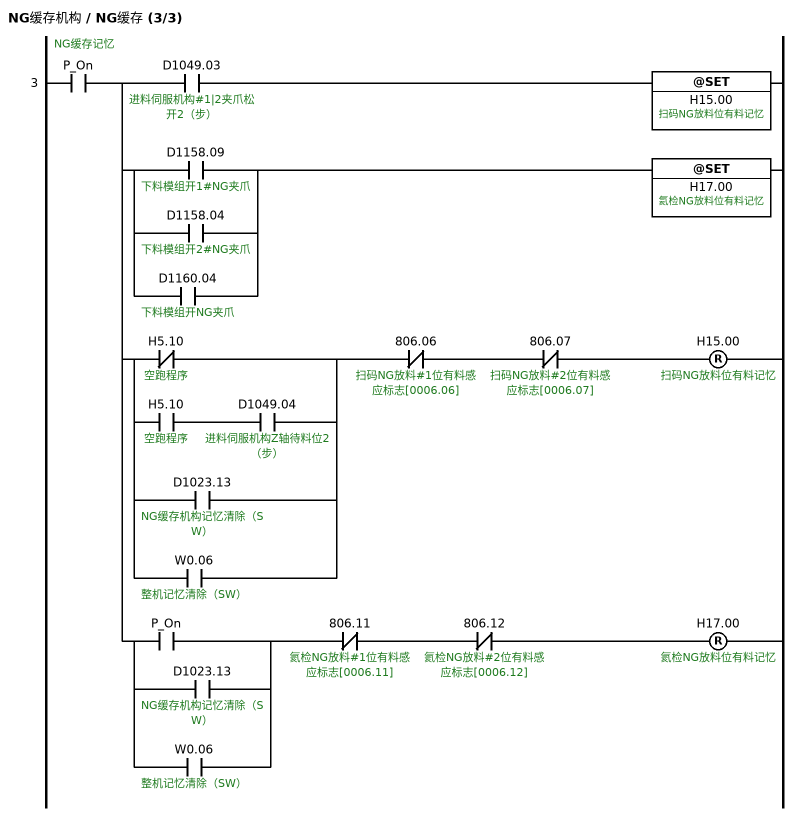
; rung 3: NG缓存记忆
LD P_On
OUT TR0
AND D1049.03  ; 进料伺服机构#1|2夹爪松开2（步）
@SET H15.00  ; 扫码NG放料位有料记忆
LD TR0
LD D1158.09  ; 下料模组开1#NG夹爪
OR D1158.04  ; 下料模组开2#NG夹爪
OR D1160.04  ; 下料模组开NG夹爪
ANDLD
@SET H17.00  ; 氦检NG放料位有料记忆
LD TR0
LDNOT H5.10  ; 空跑程序
LD H5.10  ; 空跑程序
AND D1049.04  ; 进料伺服机构Z轴待料位2（步）
ORLD
OR D1023.13  ; NG缓存机构记忆清除（SW）
OR W0.06  ; 整机记忆清除（SW）
ANDLD
ANDNOT 806.06  ; 扫码NG放料#1位有料感应标志[0006.06]
ANDNOT 806.07  ; 扫码NG放料#2位有料感应标志[0006.07]
RSET H15.00  ; 扫码NG放料位有料记忆
LD TR0
LD P_On
OR D1023.13  ; NG缓存机构记忆清除（SW）
OR W0.06  ; 整机记忆清除（SW）
ANDLD
ANDNOT 806.11  ; 氦检NG放料#1位有料感应标志[0006.11]
ANDNOT 806.12  ; 氦检NG放料#2位有料感应标志[0006.12]
RSET H17.00  ; 氦检NG放料位有料记忆

### Section 外部输出

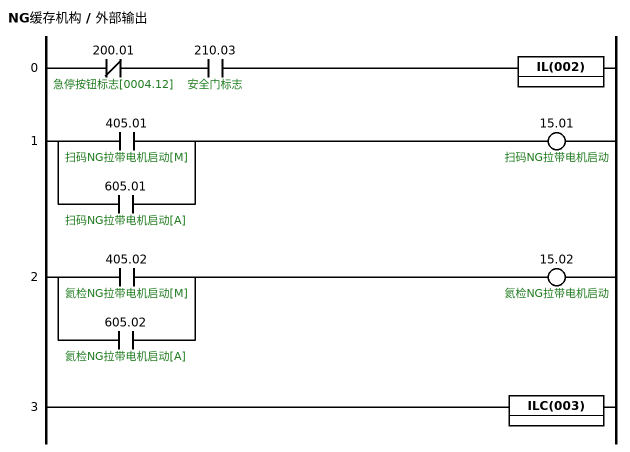
; rung 0
LDNOT 200.01  ; 急停按钮标志[0004.12]
AND 210.03  ; 安全门标志
IL(002)
; rung 1
LD 405.01  ; 扫码NG拉带电机启动[M]
OR 605.01  ; 扫码NG拉带电机启动[A]
OUT 15.01  ; 扫码NG拉带电机启动
; rung 2
LD 405.02  ; 氦检NG拉带电机启动[M]
OR 605.02  ; 氦检NG拉带电机启动[A]
OUT 15.02  ; 氦检NG拉带电机启动
; rung 3
ILC(003)

### Section END
; rung 0
END(001)

## Program Common (cyclic task 6)

### Section 动作延时

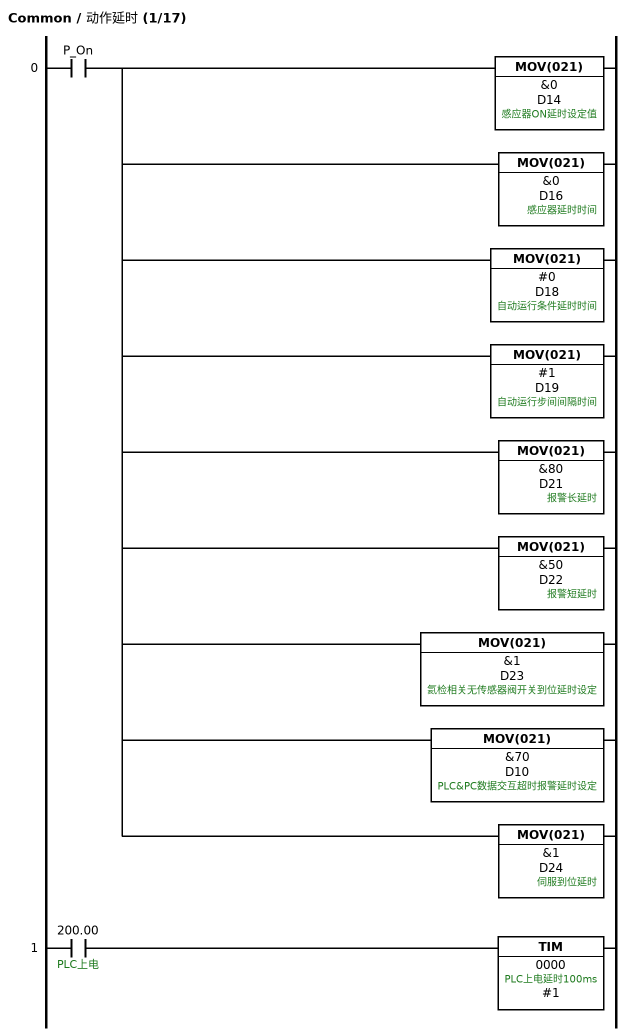
; rung 0
LD P_On
MOV(021) &0 D14  ; 感应器ON延时设定值
MOV(021) &0 D16  ; 感应器延时时间
MOV(021) #0 D18  ; 自动运行条件延时时间
MOV(021) #1 D19  ; 自动运行步间间隔时间
MOV(021) &80 D21  ; 报警长延时
MOV(021) &50 D22  ; 报警短延时
MOV(021) &1 D23  ; 氦检相关无传感器阀开关到位延时设定
MOV(021) &70 D10  ; PLC&PC数据交互超时报警延时设定
MOV(021) &1 D24  ; 伺服到位延时
; rung 1
LD 200.00  ; PLC上电
TIM 0000 #1  ; PLC上电延时100ms

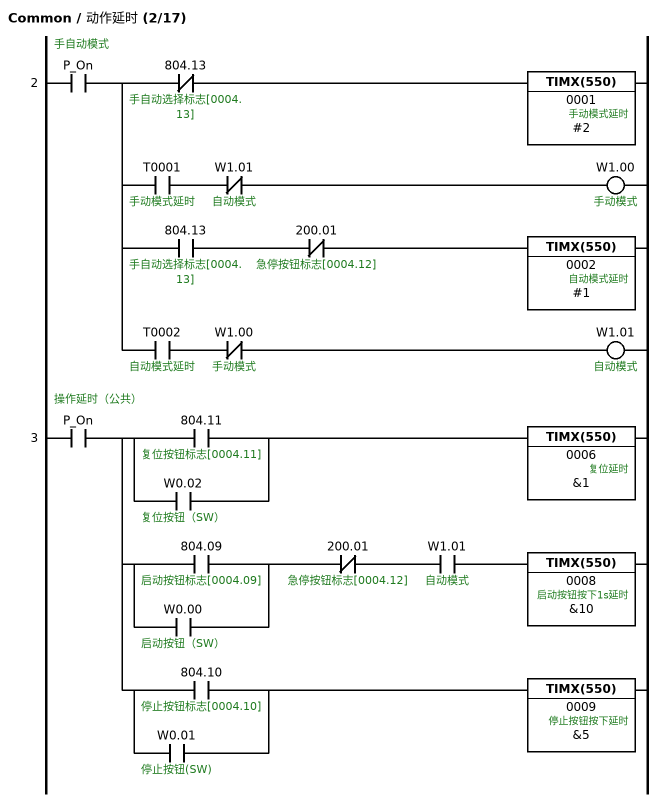
; rung 2: 手自动模式
LD P_On
OUT TR0
ANDNOT 804.13  ; 手自动选择标志[0004.13]
TIMX(550) 0001 #2  ; 手动模式延时
LD TR0
AND T0001  ; 手动模式延时
ANDNOT W1.01  ; 自动模式
OUT W1.00  ; 手动模式
LD TR0
AND 804.13  ; 手自动选择标志[0004.13]
ANDNOT 200.01  ; 急停按钮标志[0004.12]
TIMX(550) 0002 #1  ; 自动模式延时
LD TR0
AND T0002  ; 自动模式延时
ANDNOT W1.00  ; 手动模式
OUT W1.01  ; 自动模式
; rung 3: 操作延时（公共）
LD P_On
OUT TR0
LD 804.11  ; 复位按钮标志[0004.11]
OR W0.02  ; 复位按钮（SW）
ANDLD
TIMX(550) 0006 &1  ; 复位延时
LD TR0
LD 804.09  ; 启动按钮标志[0004.09]
OR W0.00  ; 启动按钮（SW）
ANDLD
ANDNOT 200.01  ; 急停按钮标志[0004.12]
AND W1.01  ; 自动模式
TIMX(550) 0008 &10  ; 启动按钮按下1s延时
LD TR0
LD 804.10  ; 停止按钮标志[0004.10]
OR W0.01  ; 停止按钮(SW)
ANDLD
TIMX(550) 0009 &5  ; 停止按钮按下延时

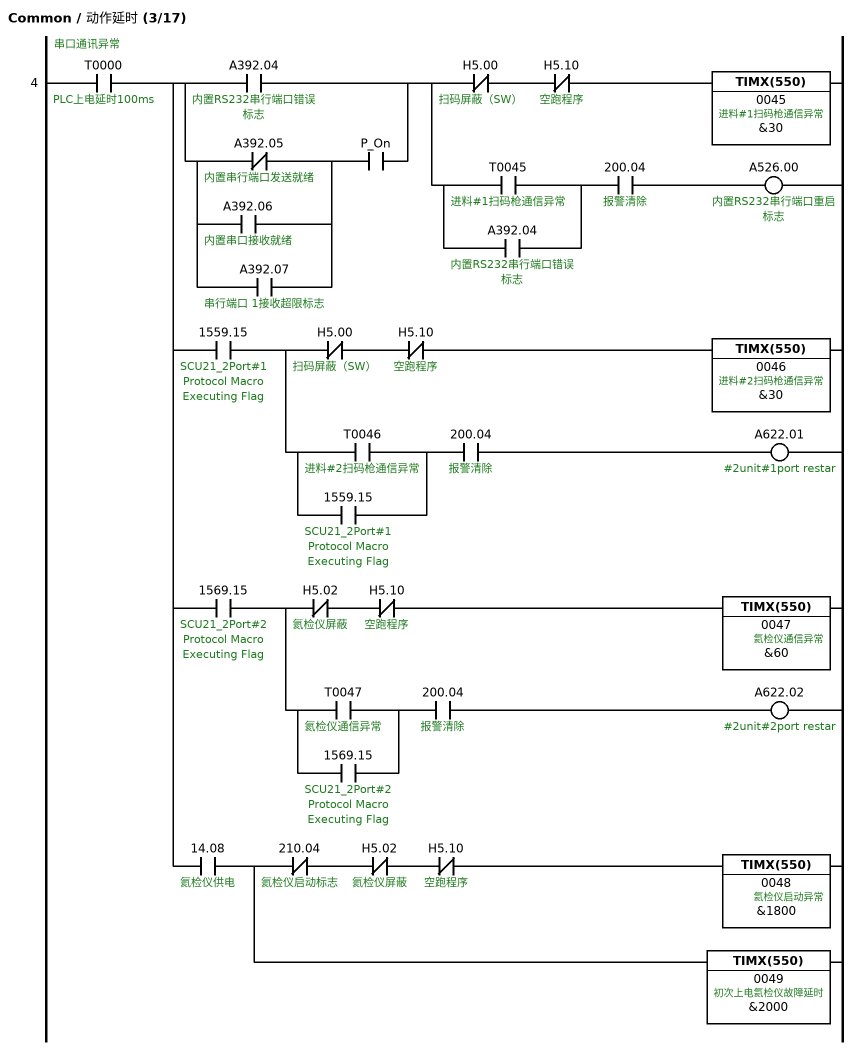
; rung 4: 串口通讯异常
LD T0000  ; PLC上电延时100ms
OUT TR0
LD A392.04  ; 内置RS232串行端口错误标志
LDNOT A392.05  ; 内置串行端口发送就绪
OR A392.06  ; 内置串口接收就绪
OR A392.07  ; 串行端口 1接收超限标志
AND P_On
ORLD
ANDLD
OUT TR1
ANDNOT H5.00  ; 扫码屏蔽（SW）
ANDNOT H5.10  ; 空跑程序
TIMX(550) 0045 &30  ; 进料#1扫码枪通信异常
LD TR1
LD T0045  ; 进料#1扫码枪通信异常
OR A392.04  ; 内置RS232串行端口错误标志
ANDLD
AND 200.04  ; 报警清除
OUT A526.00  ; 内置RS232串行端口重启标志
LD TR0
AND 1559.15  ; SCU21_2Port#1 Protocol Macro Executing Flag
OUT TR1
ANDNOT H5.00  ; 扫码屏蔽（SW）
ANDNOT H5.10  ; 空跑程序
TIMX(550) 0046 &30  ; 进料#2扫码枪通信异常
LD TR1
LD T0046  ; 进料#2扫码枪通信异常
OR 1559.15  ; SCU21_2Port#1 Protocol Macro Executing Flag
ANDLD
AND 200.04  ; 报警清除
OUT A622.01  ; #2unit#1port restar
LD TR0
AND 1569.15  ; SCU21_2Port#2 Protocol Macro Executing Flag
OUT TR1
ANDNOT H5.02  ; 氦检仪屏蔽
ANDNOT H5.10  ; 空跑程序
TIMX(550) 0047 &60  ; 氦检仪通信异常
LD TR1
LD T0047  ; 氦检仪通信异常
OR 1569.15  ; SCU21_2Port#2 Protocol Macro Executing Flag
ANDLD
AND 200.04  ; 报警清除
OUT A622.02  ; #2unit#2port restar
LD TR0
AND 14.08  ; 氦检仪供电
OUT TR0
ANDNOT 210.04  ; 氦检仪启动标志
ANDNOT H5.02  ; 氦检仪屏蔽
ANDNOT H5.10  ; 空跑程序
TIMX(550) 0048 &1800  ; 氦检仪启动异常
LD TR0
TIMX(550) 0049 &2000  ; 初次上电氦检仪故障延时
; rung 5: AI断线检测

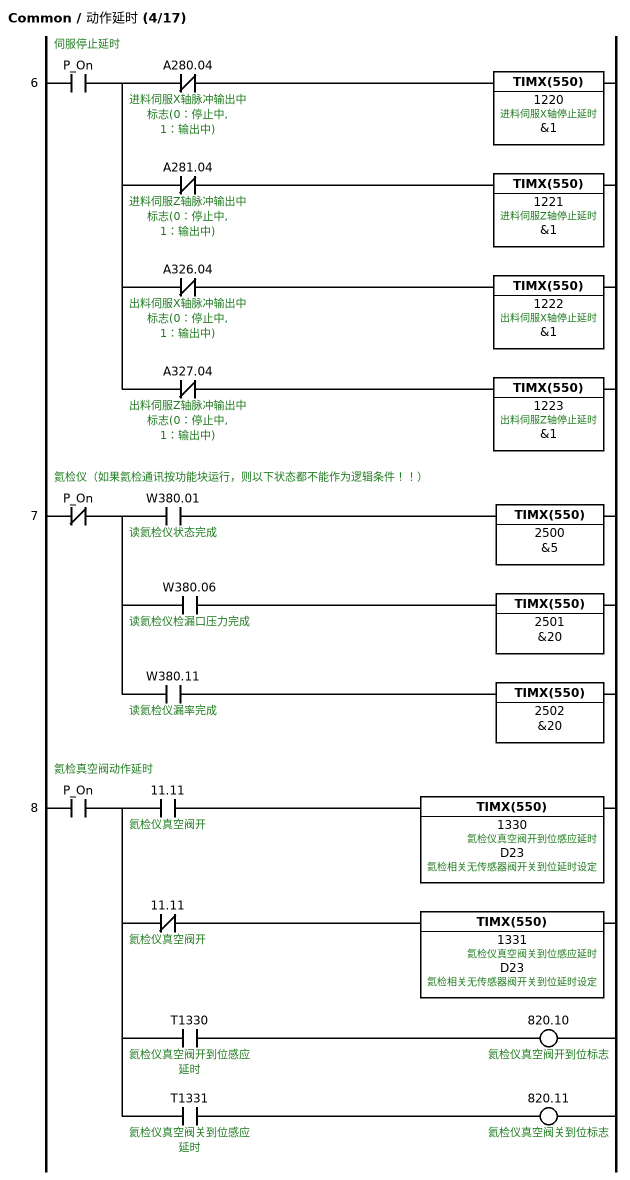
; rung 6: 伺服停止延时
LD P_On
OUT TR0
ANDNOT A280.04  ; 进料伺服X轴脉冲输出中标志(0：停止中,1：输出中)
TIMX(550) 1220 &1  ; 进料伺服X轴停止延时
LD TR0
ANDNOT A281.04  ; 进料伺服Z轴脉冲输出中标志(0：停止中,1：输出中)
TIMX(550) 1221 &1  ; 进料伺服Z轴停止延时
LD TR0
ANDNOT A326.04  ; 出料伺服X轴脉冲输出中标志(0：停止中,1：输出中)
TIMX(550) 1222 &1  ; 出料伺服X轴停止延时
LD TR0
ANDNOT A327.04  ; 出料伺服Z轴脉冲输出中标志(0：停止中,1：输出中)
TIMX(550) 1223 &1  ; 出料伺服Z轴停止延时
; rung 7: 氦检仪（如果氦检通讯按功能块运行，则以下状态都不能作为逻辑条件！！）
LDNOT P_On
OUT TR0
AND W380.01  ; 读氦检仪状态完成
TIMX(550) 2500 &5
LD TR0
AND W380.06  ; 读氦检仪检漏口压力完成
TIMX(550) 2501 &20
LD TR0
AND W380.11  ; 读氦检仪漏率完成
TIMX(550) 2502 &20
; rung 8: 氦检真空阀动作延时
LD P_On
OUT TR0
AND 11.11  ; 氦检仪真空阀开
TIMX(550) 1330 D23  ; 氦检相关无传感器阀开关到位延时设定, 氦检仪真空阀开到位感应延时
LD TR0
ANDNOT 11.11  ; 氦检仪真空阀开
TIMX(550) 1331 D23  ; 氦检相关无传感器阀开关到位延时设定, 氦检仪真空阀关到位感应延时
LD TR0
AND T1330  ; 氦检仪真空阀开到位感应延时
OUT 820.10  ; 氦检仪真空阀开到位标志
LD TR0
AND T1331  ; 氦检仪真空阀关到位感应延时
OUT 820.11  ; 氦检仪真空阀关到位标志

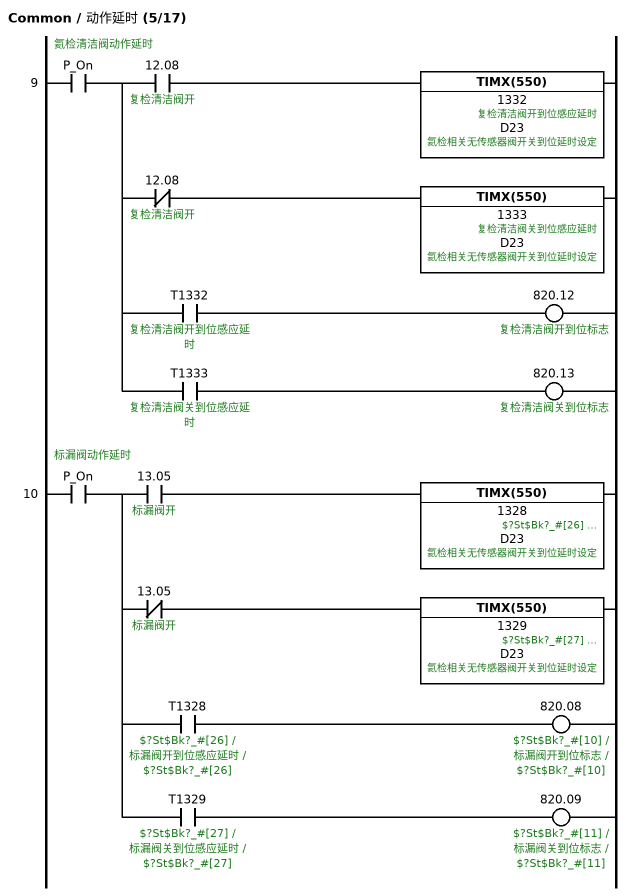
; rung 9: 氦检清洁阀动作延时
LD P_On
OUT TR0
AND 12.08  ; 复检清洁阀开
TIMX(550) 1332 D23  ; 氦检相关无传感器阀开关到位延时设定, 复检清洁阀开到位感应延时
LD TR0
ANDNOT 12.08  ; 复检清洁阀开
TIMX(550) 1333 D23  ; 氦检相关无传感器阀开关到位延时设定, 复检清洁阀关到位感应延时
LD TR0
AND T1332  ; 复检清洁阀开到位感应延时
OUT 820.12  ; 复检清洁阀开到位标志
LD TR0
AND T1333  ; 复检清洁阀关到位感应延时
OUT 820.13  ; 复检清洁阀关到位标志
; rung 10: 标漏阀动作延时
LD P_On
OUT TR0
AND 13.05  ; 标漏阀开
TIMX(550) 1328 D23  ; 氦检相关无传感器阀开关到位延时设定, $?St$Bk?_#[26] / 标漏阀开到位感应延时 / $?St$Bk?_#[26]
LD TR0
ANDNOT 13.05  ; 标漏阀开
TIMX(550) 1329 D23  ; 氦检相关无传感器阀开关到位延时设定, $?St$Bk?_#[27] / 标漏阀关到位感应延时 / $?St$Bk?_#[27]
LD TR0
AND T1328  ; $?St$Bk?_#[26] / 标漏阀开到位感应延时 / $?St$Bk?_#[26]
OUT 820.08  ; $?St$Bk?_#[10] / 标漏阀开到位标志 / $?St$Bk?_#[10]
LD TR0
AND T1329  ; $?St$Bk?_#[27] / 标漏阀关到位感应延时 / $?St$Bk?_#[27]
OUT 820.09  ; $?St$Bk?_#[11] / 标漏阀关到位标志 / $?St$Bk?_#[11]

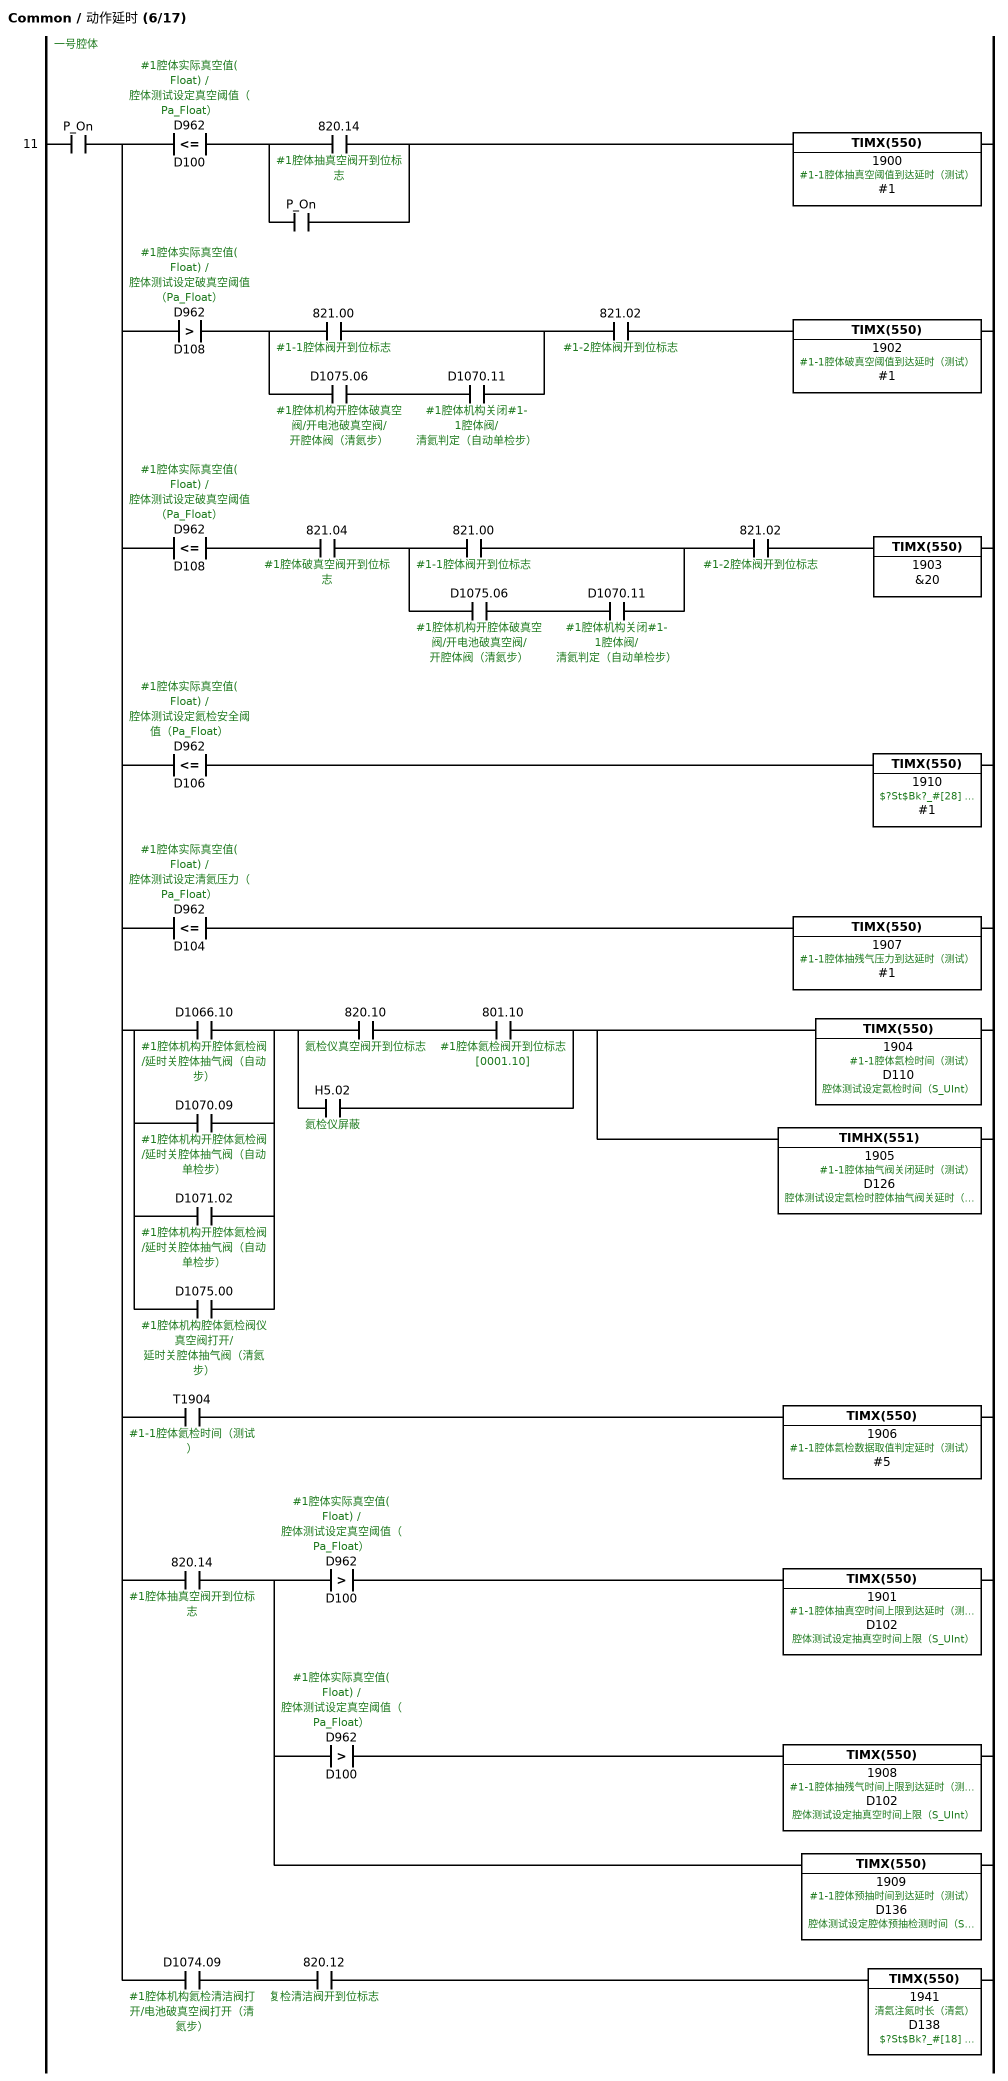
; rung 11: 一号腔体
LD P_On
OUT TR0
AND<=F(332) D962 D100  ; #1腔体实际真空值(Float), 腔体测试设定真空阈值（Pa_Float）
LD 820.14  ; #1腔体抽真空阀开到位标志
OR P_On
ANDLD
TIMX(550) 1900 #1  ; #1-1腔体抽真空阈值到达延时（测试）
LD TR0
AND>F(333) D962 D108  ; #1腔体实际真空值(Float), 腔体测试设定破真空阈值（Pa_Float）
LD 821.00  ; #1-1腔体阀开到位标志
LD D1075.06  ; #1腔体机构开腔体破真空阀/开电池破真空阀/开腔体阀（清氦步）
AND D1070.11  ; #1腔体机构关闭#1-1腔体阀/清氦判定（自动单检步）
ORLD
ANDLD
AND 821.02  ; #1-2腔体阀开到位标志
TIMX(550) 1902 #1  ; #1-1腔体破真空阈值到达延时（测试）
LD TR0
AND<=F(332) D962 D108  ; #1腔体实际真空值(Float), 腔体测试设定破真空阈值（Pa_Float）
AND 821.04  ; #1腔体破真空阀开到位标志
LD 821.00  ; #1-1腔体阀开到位标志
LD D1075.06  ; #1腔体机构开腔体破真空阀/开电池破真空阀/开腔体阀（清氦步）
AND D1070.11  ; #1腔体机构关闭#1-1腔体阀/清氦判定（自动单检步）
ORLD
ANDLD
AND 821.02  ; #1-2腔体阀开到位标志
TIMX(550) 1903 &20
LD TR0
AND<=F(332) D962 D106  ; #1腔体实际真空值(Float), 腔体测试设定氦检安全阈值（Pa_Float）
TIMX(550) 1910 #1  ; $?St$Bk?_#[28] / #1-1腔体真空在可氦检状态（测试） / $?St$Bk?_#[28]
LD TR0
AND<=F(332) D962 D104  ; #1腔体实际真空值(Float), 腔体测试设定清氦压力（Pa_Float）
TIMX(550) 1907 #1  ; #1-1腔体抽残气压力到达延时（测试）
LD TR0
LD D1066.10  ; #1腔体机构开腔体氦检阀/延时关腔体抽气阀（自动步）
OR D1070.09  ; #1腔体机构开腔体氦检阀/延时关腔体抽气阀（自动单检步）
OR D1071.02  ; #1腔体机构开腔体氦检阀/延时关腔体抽气阀（自动单检步）
OR D1075.00  ; #1腔体机构腔体氦检阀仪真空阀打开/延时关腔体抽气阀（清氦步）
ANDLD
LD 820.10  ; 氦检仪真空阀开到位标志
AND 801.10  ; #1腔体氦检阀开到位标志[0001.10]
OR H5.02  ; 氦检仪屏蔽
ANDLD
TIMX(550) 1904 D110  ; 腔体测试设定氦检时间（S_UInt）, #1-1腔体氦检时间（测试）
TIMHX(551) 1905 D126  ; 腔体测试设定氦检时腔体抽气阀关延时（S_UInt）, #1-1腔体抽气阀关闭延时（测试）
LD TR0
AND T1904  ; #1-1腔体氦检时间（测试）
TIMX(550) 1906 #5  ; #1-1腔体氦检数据取值判定延时（测试）
LD TR0
AND 820.14  ; #1腔体抽真空阀开到位标志
OUT TR1
AND>F(333) D962 D100  ; #1腔体实际真空值(Float), 腔体测试设定真空阈值（Pa_Float）
TIMX(550) 1901 D102  ; 腔体测试设定抽真空时间上限（S_UInt）, #1-1腔体抽真空时间上限到达延时（测试）
LD TR1
AND>F(333) D962 D100  ; #1腔体实际真空值(Float), 腔体测试设定真空阈值（Pa_Float）
TIMX(550) 1908 D102  ; 腔体测试设定抽真空时间上限（S_UInt）, #1-1腔体抽残气时间上限到达延时（测试）
LD TR1
TIMX(550) 1909 D136  ; 腔体测试设定腔体预抽检测时间（S_UInt）, #1-1腔体预抽时间到达延时（测试）
LD TR0
AND D1074.09  ; #1腔体机构氦检清洁阀打开/电池破真空阀打开（清氦步）
AND 820.12  ; 复检清洁阀开到位标志
TIMX(550) 1941 D138  ; $?St$Bk?_#[18] / 管路清氦注氮时间（S_UInt） / $?St$Bk?_#[18], 清氦注氮时长（清氦）

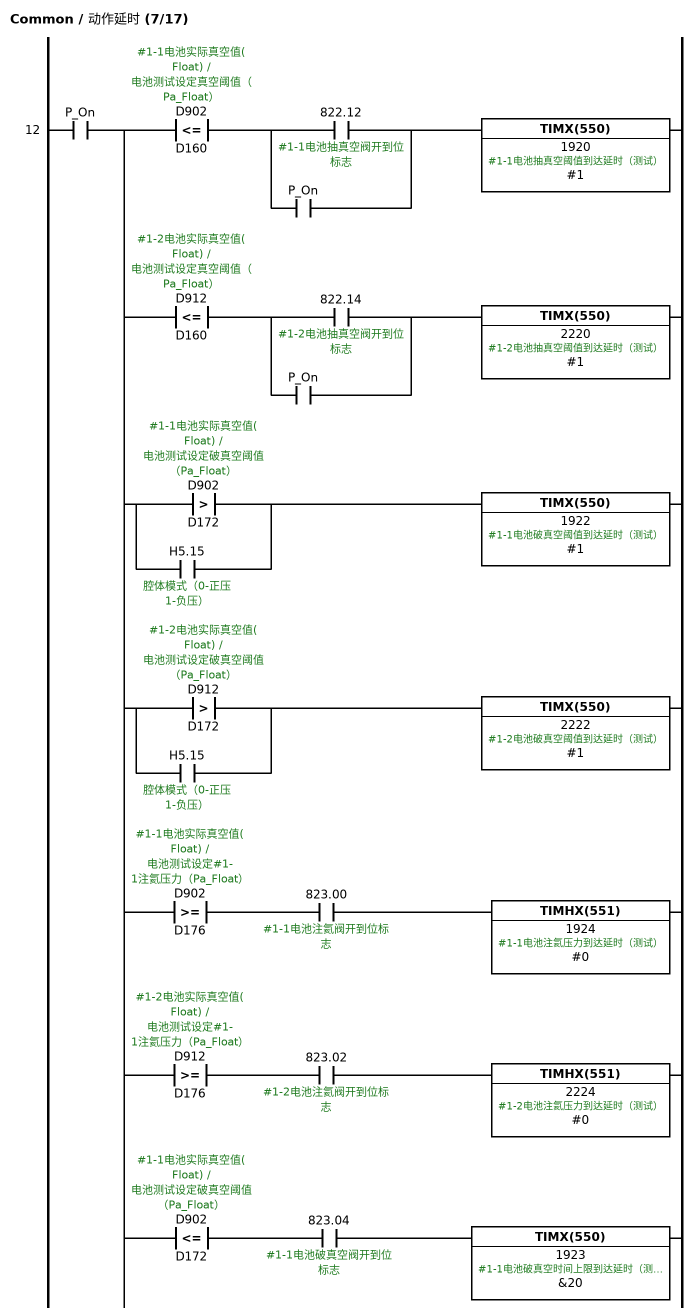

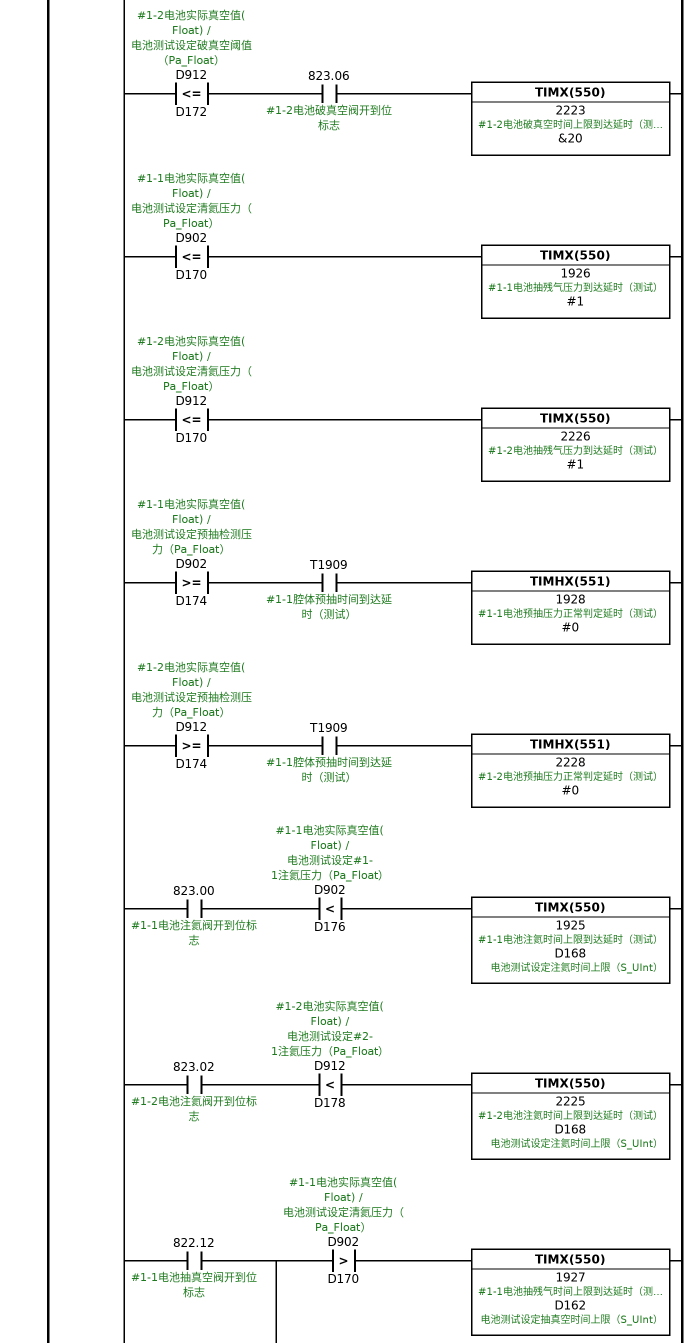

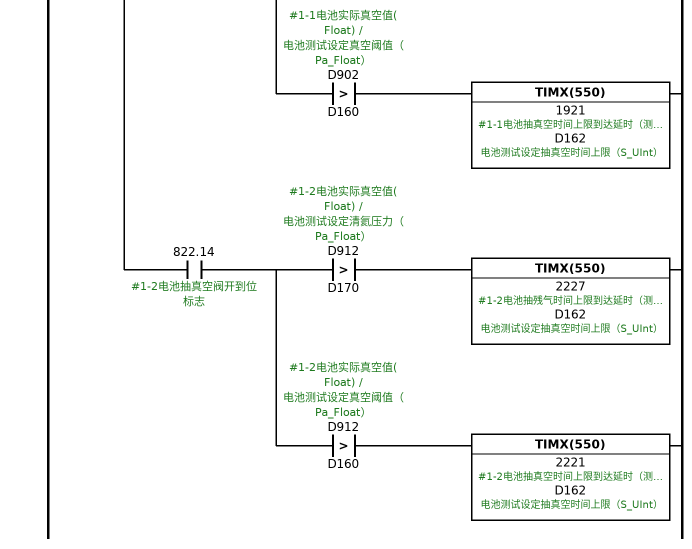
; rung 12
LD P_On
OUT TR0
AND<=F(332) D902 D160  ; #1-1电池实际真空值(Float), 电池测试设定真空阈值（Pa_Float）
LD 822.12  ; #1-1电池抽真空阀开到位标志
OR P_On
ANDLD
TIMX(550) 1920 #1  ; #1-1电池抽真空阈值到达延时（测试）
LD TR0
AND<=F(332) D912 D160  ; #1-2电池实际真空值(Float), 电池测试设定真空阈值（Pa_Float）
LD 822.14  ; #1-2电池抽真空阀开到位标志
OR P_On
ANDLD
TIMX(550) 2220 #1  ; #1-2电池抽真空阈值到达延时（测试）
LD TR0
LD>F(333) D902 D172  ; #1-1电池实际真空值(Float), 电池测试设定破真空阈值（Pa_Float）
OR H5.15  ; 腔体模式（0-正压 1-负压）
ANDLD
TIMX(550) 1922 #1  ; #1-1电池破真空阈值到达延时（测试）
LD TR0
LD>F(333) D912 D172  ; #1-2电池实际真空值(Float), 电池测试设定破真空阈值（Pa_Float）
OR H5.15  ; 腔体模式（0-正压 1-负压）
ANDLD
TIMX(550) 2222 #1  ; #1-2电池破真空阈值到达延时（测试）
LD TR0
AND>=F(334) D902 D176  ; #1-1电池实际真空值(Float), 电池测试设定#1-1注氦压力（Pa_Float）
AND 823.00  ; #1-1电池注氦阀开到位标志
TIMHX(551) 1924 #0  ; #1-1电池注氦压力到达延时（测试）
LD TR0
AND>=F(334) D912 D176  ; #1-2电池实际真空值(Float), 电池测试设定#1-1注氦压力（Pa_Float）
AND 823.02  ; #1-2电池注氦阀开到位标志
TIMHX(551) 2224 #0  ; #1-2电池注氦压力到达延时（测试）
LD TR0
AND<=F(332) D902 D172  ; #1-1电池实际真空值(Float), 电池测试设定破真空阈值（Pa_Float）
AND 823.04  ; #1-1电池破真空阀开到位标志
TIMX(550) 1923 &20  ; #1-1电池破真空时间上限到达延时（测试）
LD TR0
AND<=F(332) D912 D172  ; #1-2电池实际真空值(Float), 电池测试设定破真空阈值（Pa_Float）
AND 823.06  ; #1-2电池破真空阀开到位标志
TIMX(550) 2223 &20  ; #1-2电池破真空时间上限到达延时（测试）
LD TR0
AND<=F(332) D902 D170  ; #1-1电池实际真空值(Float), 电池测试设定清氦压力（Pa_Float）
TIMX(550) 1926 #1  ; #1-1电池抽残气压力到达延时（测试）
LD TR0
AND<=F(332) D912 D170  ; #1-2电池实际真空值(Float), 电池测试设定清氦压力（Pa_Float）
TIMX(550) 2226 #1  ; #1-2电池抽残气压力到达延时（测试）
LD TR0
AND>=F(334) D902 D174  ; #1-1电池实际真空值(Float), 电池测试设定预抽检测压力（Pa_Float）
AND T1909  ; #1-1腔体预抽时间到达延时（测试）
TIMHX(551) 1928 #0  ; #1-1电池预抽压力正常判定延时（测试）
LD TR0
AND>=F(334) D912 D174  ; #1-2电池实际真空值(Float), 电池测试设定预抽检测压力（Pa_Float）
AND T1909  ; #1-1腔体预抽时间到达延时（测试）
TIMHX(551) 2228 #0  ; #1-2电池预抽压力正常判定延时（测试）
LD TR0
AND 823.00  ; #1-1电池注氦阀开到位标志
AND<F(331) D902 D176  ; #1-1电池实际真空值(Float), 电池测试设定#1-1注氦压力（Pa_Float）
TIMX(550) 1925 D168  ; 电池测试设定注氦时间上限（S_UInt）, #1-1电池注氦时间上限到达延时（测试）
LD TR0
AND 823.02  ; #1-2电池注氦阀开到位标志
AND<F(331) D912 D178  ; #1-2电池实际真空值(Float), 电池测试设定#2-1注氦压力（Pa_Float）
TIMX(550) 2225 D168  ; 电池测试设定注氦时间上限（S_UInt）, #1-2电池注氦时间上限到达延时（测试）
LD TR0
AND 822.12  ; #1-1电池抽真空阀开到位标志
OUT TR1
AND>F(333) D902 D170  ; #1-1电池实际真空值(Float), 电池测试设定清氦压力（Pa_Float）
TIMX(550) 1927 D162  ; 电池测试设定抽真空时间上限（S_UInt）, #1-1电池抽残气时间上限到达延时（测试）
LD TR1
AND>F(333) D902 D160  ; #1-1电池实际真空值(Float), 电池测试设定真空阈值（Pa_Float）
TIMX(550) 1921 D162  ; 电池测试设定抽真空时间上限（S_UInt）, #1-1电池抽真空时间上限到达延时（测试）
LD TR0
AND 822.14  ; #1-2电池抽真空阀开到位标志
OUT TR0
AND>F(333) D912 D170  ; #1-2电池实际真空值(Float), 电池测试设定清氦压力（Pa_Float）
TIMX(550) 2227 D162  ; 电池测试设定抽真空时间上限（S_UInt）, #1-2电池抽残气时间上限到达延时（测试）
LD TR0
AND>F(333) D912 D160  ; #1-2电池实际真空值(Float), 电池测试设定真空阈值（Pa_Float）
TIMX(550) 2221 D162  ; 电池测试设定抽真空时间上限（S_UInt）, #1-2电池抽真空时间上限到达延时（测试）

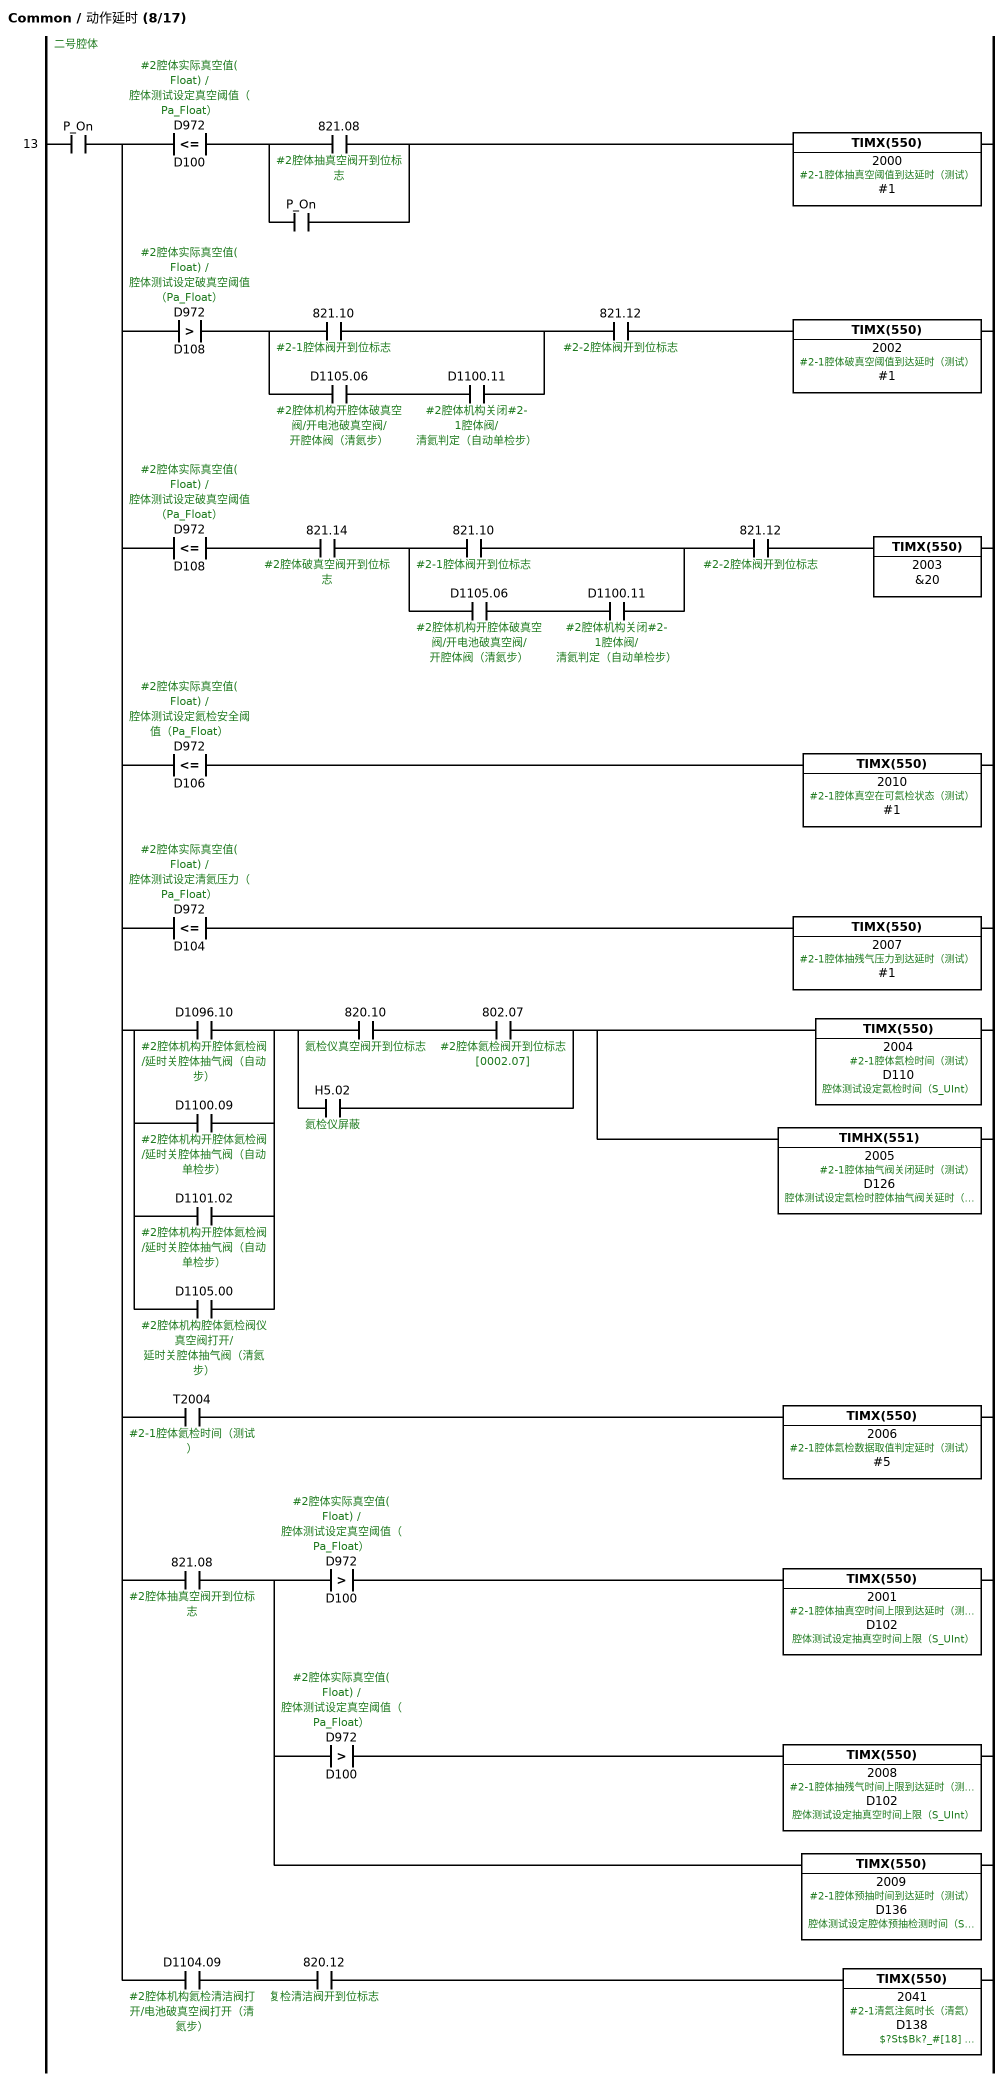
; rung 13: 二号腔体
LD P_On
OUT TR0
AND<=F(332) D972 D100  ; #2腔体实际真空值(Float), 腔体测试设定真空阈值（Pa_Float）
LD 821.08  ; #2腔体抽真空阀开到位标志
OR P_On
ANDLD
TIMX(550) 2000 #1  ; #2-1腔体抽真空阈值到达延时（测试）
LD TR0
AND>F(333) D972 D108  ; #2腔体实际真空值(Float), 腔体测试设定破真空阈值（Pa_Float）
LD 821.10  ; #2-1腔体阀开到位标志
LD D1105.06  ; #2腔体机构开腔体破真空阀/开电池破真空阀/开腔体阀（清氦步）
AND D1100.11  ; #2腔体机构关闭#2-1腔体阀/清氦判定（自动单检步）
ORLD
ANDLD
AND 821.12  ; #2-2腔体阀开到位标志
TIMX(550) 2002 #1  ; #2-1腔体破真空阈值到达延时（测试）
LD TR0
AND<=F(332) D972 D108  ; #2腔体实际真空值(Float), 腔体测试设定破真空阈值（Pa_Float）
AND 821.14  ; #2腔体破真空阀开到位标志
LD 821.10  ; #2-1腔体阀开到位标志
LD D1105.06  ; #2腔体机构开腔体破真空阀/开电池破真空阀/开腔体阀（清氦步）
AND D1100.11  ; #2腔体机构关闭#2-1腔体阀/清氦判定（自动单检步）
ORLD
ANDLD
AND 821.12  ; #2-2腔体阀开到位标志
TIMX(550) 2003 &20
LD TR0
AND<=F(332) D972 D106  ; #2腔体实际真空值(Float), 腔体测试设定氦检安全阈值（Pa_Float）
TIMX(550) 2010 #1  ; #2-1腔体真空在可氦检状态（测试）
LD TR0
AND<=F(332) D972 D104  ; #2腔体实际真空值(Float), 腔体测试设定清氦压力（Pa_Float）
TIMX(550) 2007 #1  ; #2-1腔体抽残气压力到达延时（测试）
LD TR0
LD D1096.10  ; #2腔体机构开腔体氦检阀/延时关腔体抽气阀（自动步）
OR D1100.09  ; #2腔体机构开腔体氦检阀/延时关腔体抽气阀（自动单检步）
OR D1101.02  ; #2腔体机构开腔体氦检阀/延时关腔体抽气阀（自动单检步）
OR D1105.00  ; #2腔体机构腔体氦检阀仪真空阀打开/延时关腔体抽气阀（清氦步）
ANDLD
LD 820.10  ; 氦检仪真空阀开到位标志
AND 802.07  ; #2腔体氦检阀开到位标志[0002.07]
OR H5.02  ; 氦检仪屏蔽
ANDLD
TIMX(550) 2004 D110  ; 腔体测试设定氦检时间（S_UInt）, #2-1腔体氦检时间（测试）
TIMHX(551) 2005 D126  ; 腔体测试设定氦检时腔体抽气阀关延时（S_UInt）, #2-1腔体抽气阀关闭延时（测试）
LD TR0
AND T2004  ; #2-1腔体氦检时间（测试）
TIMX(550) 2006 #5  ; #2-1腔体氦检数据取值判定延时（测试）
LD TR0
AND 821.08  ; #2腔体抽真空阀开到位标志
OUT TR1
AND>F(333) D972 D100  ; #2腔体实际真空值(Float), 腔体测试设定真空阈值（Pa_Float）
TIMX(550) 2001 D102  ; 腔体测试设定抽真空时间上限（S_UInt）, #2-1腔体抽真空时间上限到达延时（测试）
LD TR1
AND>F(333) D972 D100  ; #2腔体实际真空值(Float), 腔体测试设定真空阈值（Pa_Float）
TIMX(550) 2008 D102  ; 腔体测试设定抽真空时间上限（S_UInt）, #2-1腔体抽残气时间上限到达延时（测试）
LD TR1
TIMX(550) 2009 D136  ; 腔体测试设定腔体预抽检测时间（S_UInt）, #2-1腔体预抽时间到达延时（测试）
LD TR0
AND D1104.09  ; #2腔体机构氦检清洁阀打开/电池破真空阀打开（清氦步）
AND 820.12  ; 复检清洁阀开到位标志
TIMX(550) 2041 D138  ; $?St$Bk?_#[18] / 管路清氦注氮时间（S_UInt） / $?St$Bk?_#[18], #2-1清氦注氮时长（清氦）

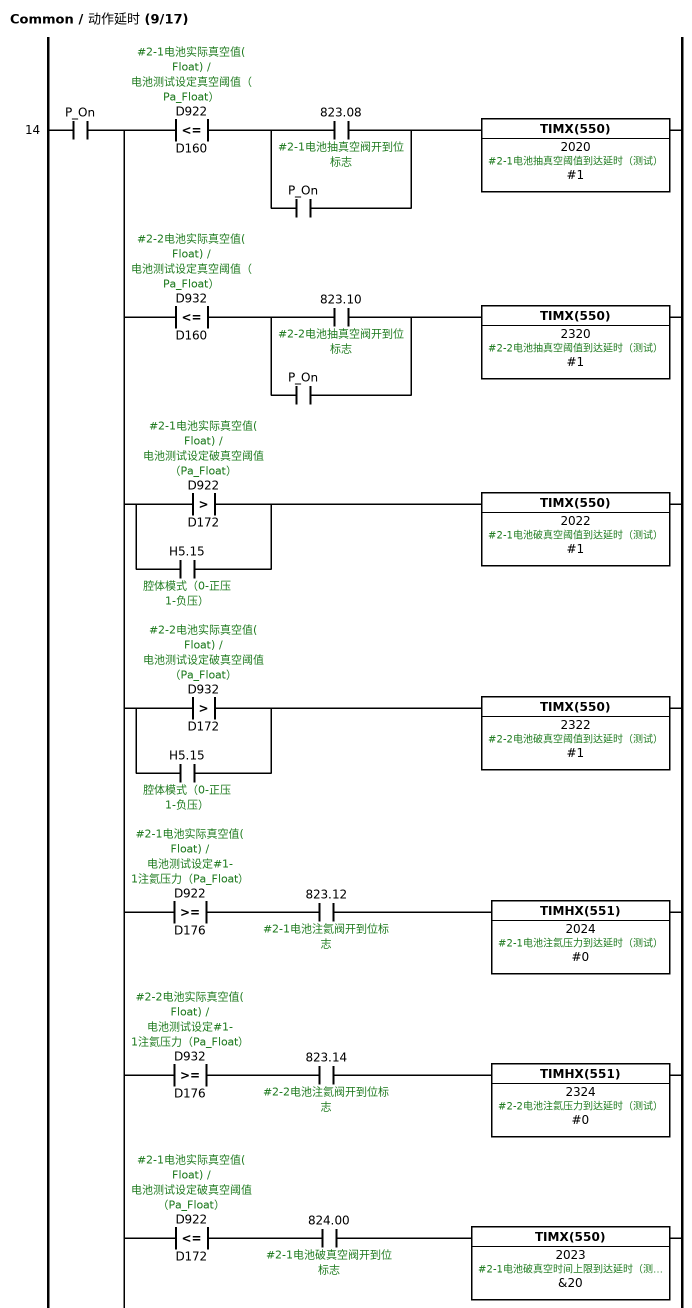

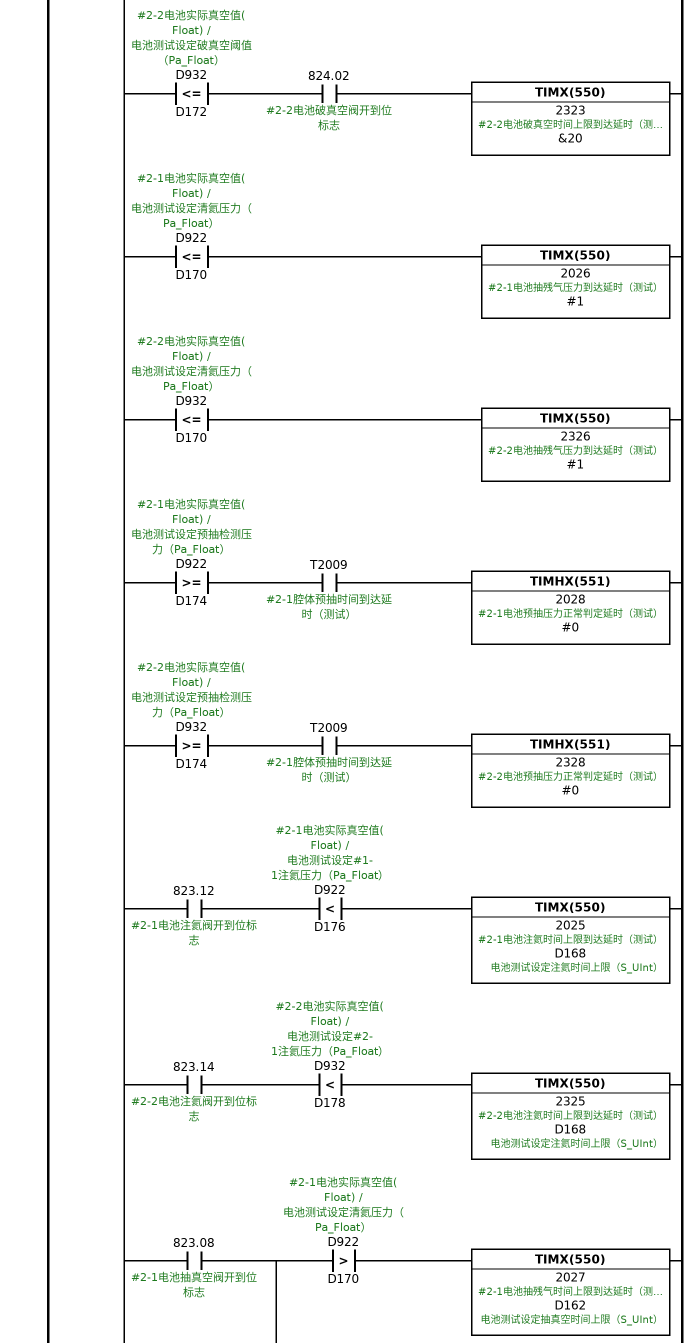

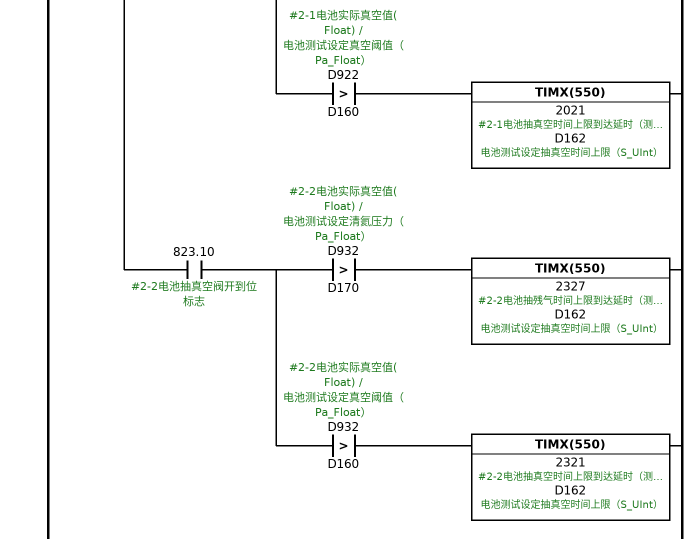
; rung 14
LD P_On
OUT TR0
AND<=F(332) D922 D160  ; #2-1电池实际真空值(Float), 电池测试设定真空阈值（Pa_Float）
LD 823.08  ; #2-1电池抽真空阀开到位标志
OR P_On
ANDLD
TIMX(550) 2020 #1  ; #2-1电池抽真空阈值到达延时（测试）
LD TR0
AND<=F(332) D932 D160  ; #2-2电池实际真空值(Float), 电池测试设定真空阈值（Pa_Float）
LD 823.10  ; #2-2电池抽真空阀开到位标志
OR P_On
ANDLD
TIMX(550) 2320 #1  ; #2-2电池抽真空阈值到达延时（测试）
LD TR0
LD>F(333) D922 D172  ; #2-1电池实际真空值(Float), 电池测试设定破真空阈值（Pa_Float）
OR H5.15  ; 腔体模式（0-正压 1-负压）
ANDLD
TIMX(550) 2022 #1  ; #2-1电池破真空阈值到达延时（测试）
LD TR0
LD>F(333) D932 D172  ; #2-2电池实际真空值(Float), 电池测试设定破真空阈值（Pa_Float）
OR H5.15  ; 腔体模式（0-正压 1-负压）
ANDLD
TIMX(550) 2322 #1  ; #2-2电池破真空阈值到达延时（测试）
LD TR0
AND>=F(334) D922 D176  ; #2-1电池实际真空值(Float), 电池测试设定#1-1注氦压力（Pa_Float）
AND 823.12  ; #2-1电池注氦阀开到位标志
TIMHX(551) 2024 #0  ; #2-1电池注氦压力到达延时（测试）
LD TR0
AND>=F(334) D932 D176  ; #2-2电池实际真空值(Float), 电池测试设定#1-1注氦压力（Pa_Float）
AND 823.14  ; #2-2电池注氦阀开到位标志
TIMHX(551) 2324 #0  ; #2-2电池注氦压力到达延时（测试）
LD TR0
AND<=F(332) D922 D172  ; #2-1电池实际真空值(Float), 电池测试设定破真空阈值（Pa_Float）
AND 824.00  ; #2-1电池破真空阀开到位标志
TIMX(550) 2023 &20  ; #2-1电池破真空时间上限到达延时（测试）
LD TR0
AND<=F(332) D932 D172  ; #2-2电池实际真空值(Float), 电池测试设定破真空阈值（Pa_Float）
AND 824.02  ; #2-2电池破真空阀开到位标志
TIMX(550) 2323 &20  ; #2-2电池破真空时间上限到达延时（测试）
LD TR0
AND<=F(332) D922 D170  ; #2-1电池实际真空值(Float), 电池测试设定清氦压力（Pa_Float）
TIMX(550) 2026 #1  ; #2-1电池抽残气压力到达延时（测试）
LD TR0
AND<=F(332) D932 D170  ; #2-2电池实际真空值(Float), 电池测试设定清氦压力（Pa_Float）
TIMX(550) 2326 #1  ; #2-2电池抽残气压力到达延时（测试）
LD TR0
AND>=F(334) D922 D174  ; #2-1电池实际真空值(Float), 电池测试设定预抽检测压力（Pa_Float）
AND T2009  ; #2-1腔体预抽时间到达延时（测试）
TIMHX(551) 2028 #0  ; #2-1电池预抽压力正常判定延时（测试）
LD TR0
AND>=F(334) D932 D174  ; #2-2电池实际真空值(Float), 电池测试设定预抽检测压力（Pa_Float）
AND T2009  ; #2-1腔体预抽时间到达延时（测试）
TIMHX(551) 2328 #0  ; #2-2电池预抽压力正常判定延时（测试）
LD TR0
AND 823.12  ; #2-1电池注氦阀开到位标志
AND<F(331) D922 D176  ; #2-1电池实际真空值(Float), 电池测试设定#1-1注氦压力（Pa_Float）
TIMX(550) 2025 D168  ; 电池测试设定注氦时间上限（S_UInt）, #2-1电池注氦时间上限到达延时（测试）
LD TR0
AND 823.14  ; #2-2电池注氦阀开到位标志
AND<F(331) D932 D178  ; #2-2电池实际真空值(Float), 电池测试设定#2-1注氦压力（Pa_Float）
TIMX(550) 2325 D168  ; 电池测试设定注氦时间上限（S_UInt）, #2-2电池注氦时间上限到达延时（测试）
LD TR0
AND 823.08  ; #2-1电池抽真空阀开到位标志
OUT TR1
AND>F(333) D922 D170  ; #2-1电池实际真空值(Float), 电池测试设定清氦压力（Pa_Float）
TIMX(550) 2027 D162  ; 电池测试设定抽真空时间上限（S_UInt）, #2-1电池抽残气时间上限到达延时（测试）
LD TR1
AND>F(333) D922 D160  ; #2-1电池实际真空值(Float), 电池测试设定真空阈值（Pa_Float）
TIMX(550) 2021 D162  ; 电池测试设定抽真空时间上限（S_UInt）, #2-1电池抽真空时间上限到达延时（测试）
LD TR0
AND 823.10  ; #2-2电池抽真空阀开到位标志
OUT TR0
AND>F(333) D932 D170  ; #2-2电池实际真空值(Float), 电池测试设定清氦压力（Pa_Float）
TIMX(550) 2327 D162  ; 电池测试设定抽真空时间上限（S_UInt）, #2-2电池抽残气时间上限到达延时（测试）
LD TR0
AND>F(333) D932 D160  ; #2-2电池实际真空值(Float), 电池测试设定真空阈值（Pa_Float）
TIMX(550) 2321 D162  ; 电池测试设定抽真空时间上限（S_UInt）, #2-2电池抽真空时间上限到达延时（测试）

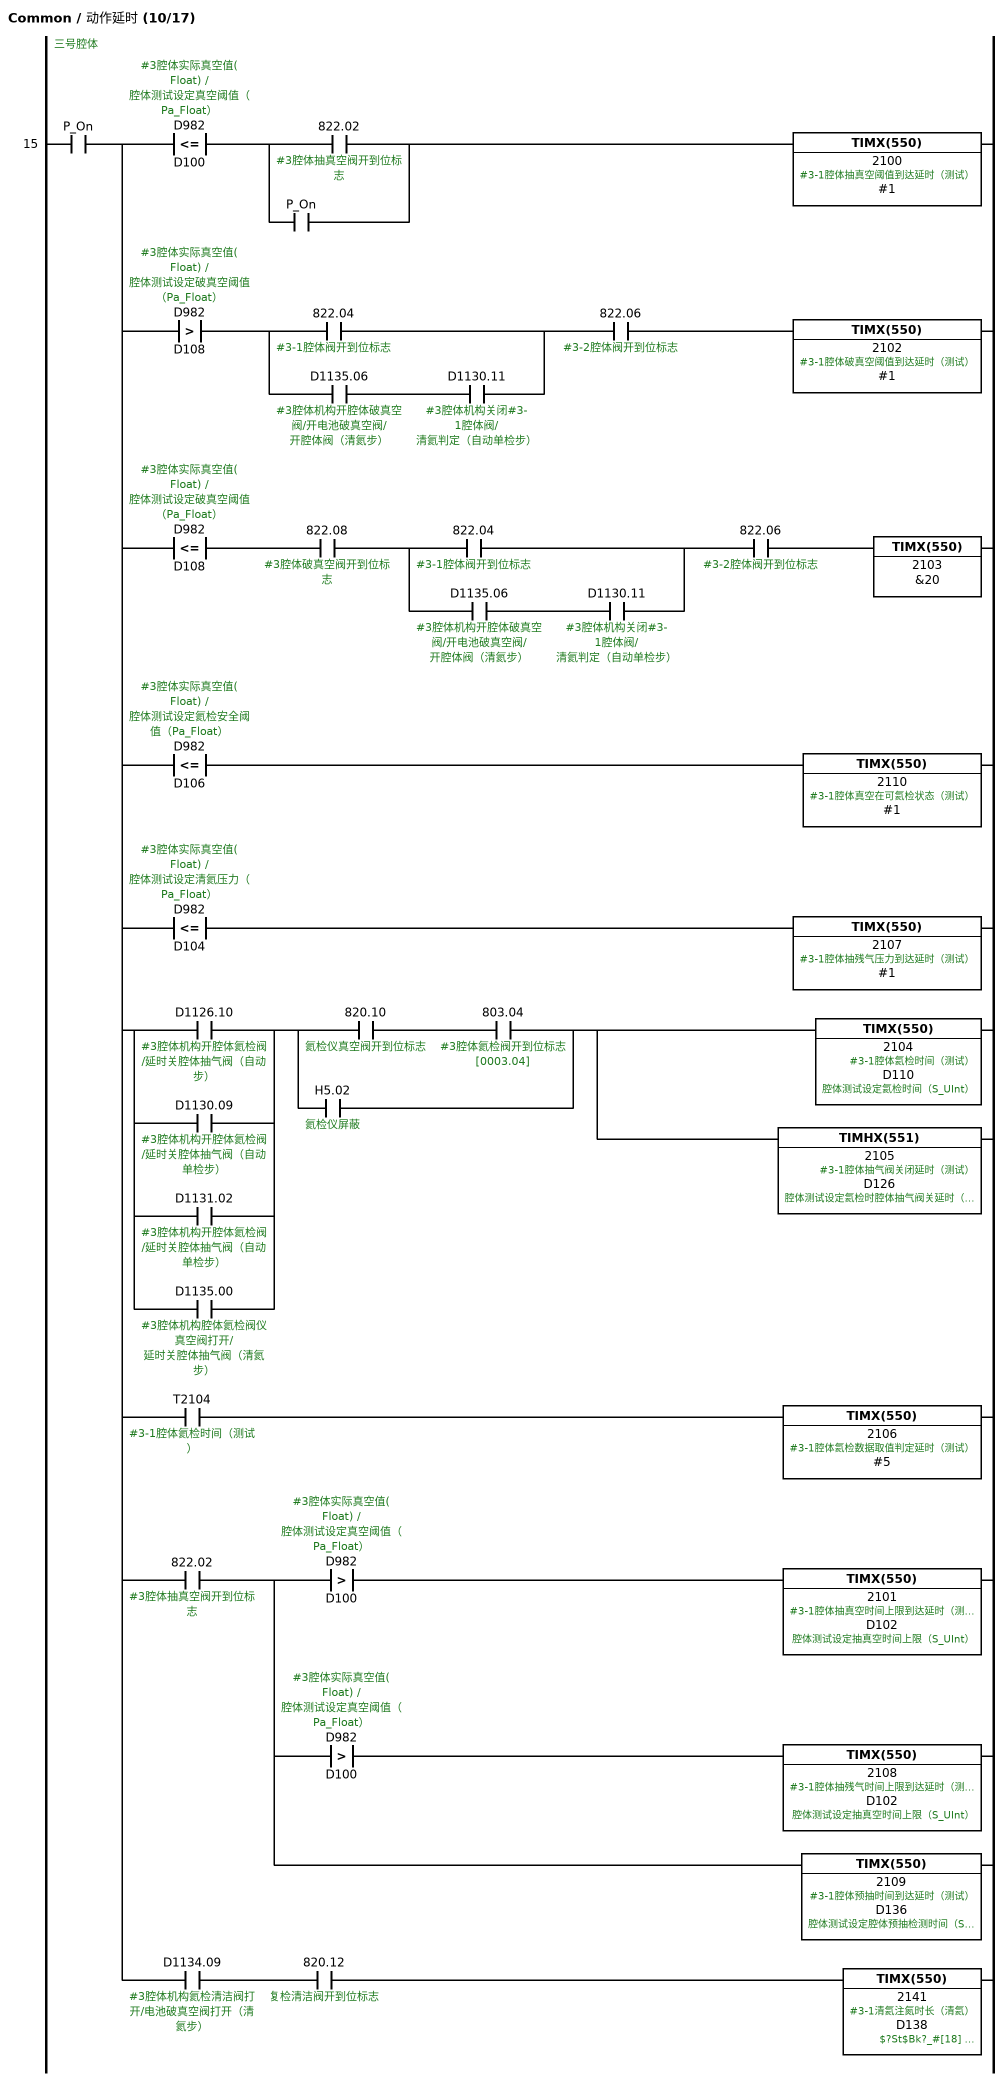
; rung 15: 三号腔体
LD P_On
OUT TR0
AND<=F(332) D982 D100  ; #3腔体实际真空值(Float), 腔体测试设定真空阈值（Pa_Float）
LD 822.02  ; #3腔体抽真空阀开到位标志
OR P_On
ANDLD
TIMX(550) 2100 #1  ; #3-1腔体抽真空阈值到达延时（测试）
LD TR0
AND>F(333) D982 D108  ; #3腔体实际真空值(Float), 腔体测试设定破真空阈值（Pa_Float）
LD 822.04  ; #3-1腔体阀开到位标志
LD D1135.06  ; #3腔体机构开腔体破真空阀/开电池破真空阀/开腔体阀（清氦步）
AND D1130.11  ; #3腔体机构关闭#3-1腔体阀/清氦判定（自动单检步）
ORLD
ANDLD
AND 822.06  ; #3-2腔体阀开到位标志
TIMX(550) 2102 #1  ; #3-1腔体破真空阈值到达延时（测试）
LD TR0
AND<=F(332) D982 D108  ; #3腔体实际真空值(Float), 腔体测试设定破真空阈值（Pa_Float）
AND 822.08  ; #3腔体破真空阀开到位标志
LD 822.04  ; #3-1腔体阀开到位标志
LD D1135.06  ; #3腔体机构开腔体破真空阀/开电池破真空阀/开腔体阀（清氦步）
AND D1130.11  ; #3腔体机构关闭#3-1腔体阀/清氦判定（自动单检步）
ORLD
ANDLD
AND 822.06  ; #3-2腔体阀开到位标志
TIMX(550) 2103 &20
LD TR0
AND<=F(332) D982 D106  ; #3腔体实际真空值(Float), 腔体测试设定氦检安全阈值（Pa_Float）
TIMX(550) 2110 #1  ; #3-1腔体真空在可氦检状态（测试）
LD TR0
AND<=F(332) D982 D104  ; #3腔体实际真空值(Float), 腔体测试设定清氦压力（Pa_Float）
TIMX(550) 2107 #1  ; #3-1腔体抽残气压力到达延时（测试）
LD TR0
LD D1126.10  ; #3腔体机构开腔体氦检阀/延时关腔体抽气阀（自动步）
OR D1130.09  ; #3腔体机构开腔体氦检阀/延时关腔体抽气阀（自动单检步）
OR D1131.02  ; #3腔体机构开腔体氦检阀/延时关腔体抽气阀（自动单检步）
OR D1135.00  ; #3腔体机构腔体氦检阀仪真空阀打开/延时关腔体抽气阀（清氦步）
ANDLD
LD 820.10  ; 氦检仪真空阀开到位标志
AND 803.04  ; #3腔体氦检阀开到位标志[0003.04]
OR H5.02  ; 氦检仪屏蔽
ANDLD
TIMX(550) 2104 D110  ; 腔体测试设定氦检时间（S_UInt）, #3-1腔体氦检时间（测试）
TIMHX(551) 2105 D126  ; 腔体测试设定氦检时腔体抽气阀关延时（S_UInt）, #3-1腔体抽气阀关闭延时（测试）
LD TR0
AND T2104  ; #3-1腔体氦检时间（测试）
TIMX(550) 2106 #5  ; #3-1腔体氦检数据取值判定延时（测试）
LD TR0
AND 822.02  ; #3腔体抽真空阀开到位标志
OUT TR1
AND>F(333) D982 D100  ; #3腔体实际真空值(Float), 腔体测试设定真空阈值（Pa_Float）
TIMX(550) 2101 D102  ; 腔体测试设定抽真空时间上限（S_UInt）, #3-1腔体抽真空时间上限到达延时（测试）
LD TR1
AND>F(333) D982 D100  ; #3腔体实际真空值(Float), 腔体测试设定真空阈值（Pa_Float）
TIMX(550) 2108 D102  ; 腔体测试设定抽真空时间上限（S_UInt）, #3-1腔体抽残气时间上限到达延时（测试）
LD TR1
TIMX(550) 2109 D136  ; 腔体测试设定腔体预抽检测时间（S_UInt）, #3-1腔体预抽时间到达延时（测试）
LD TR0
AND D1134.09  ; #3腔体机构氦检清洁阀打开/电池破真空阀打开（清氦步）
AND 820.12  ; 复检清洁阀开到位标志
TIMX(550) 2141 D138  ; $?St$Bk?_#[18] / 管路清氦注氮时间（S_UInt） / $?St$Bk?_#[18], #3-1清氦注氮时长（清氦）

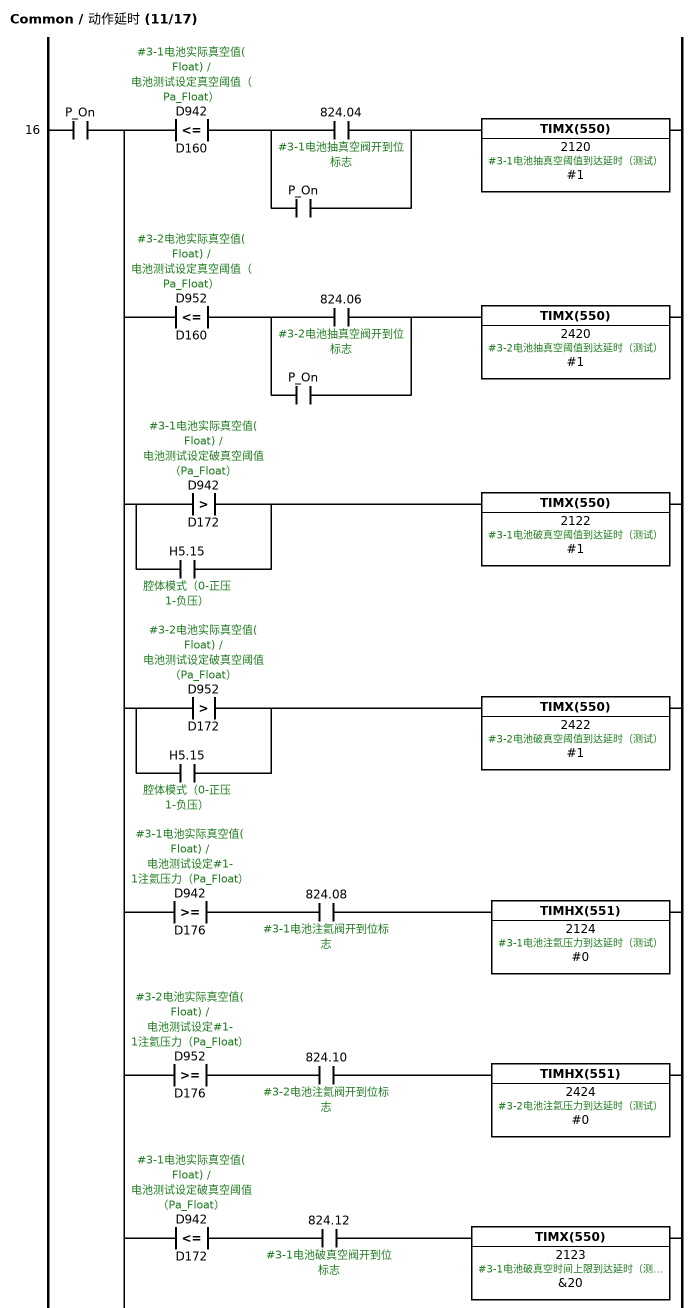

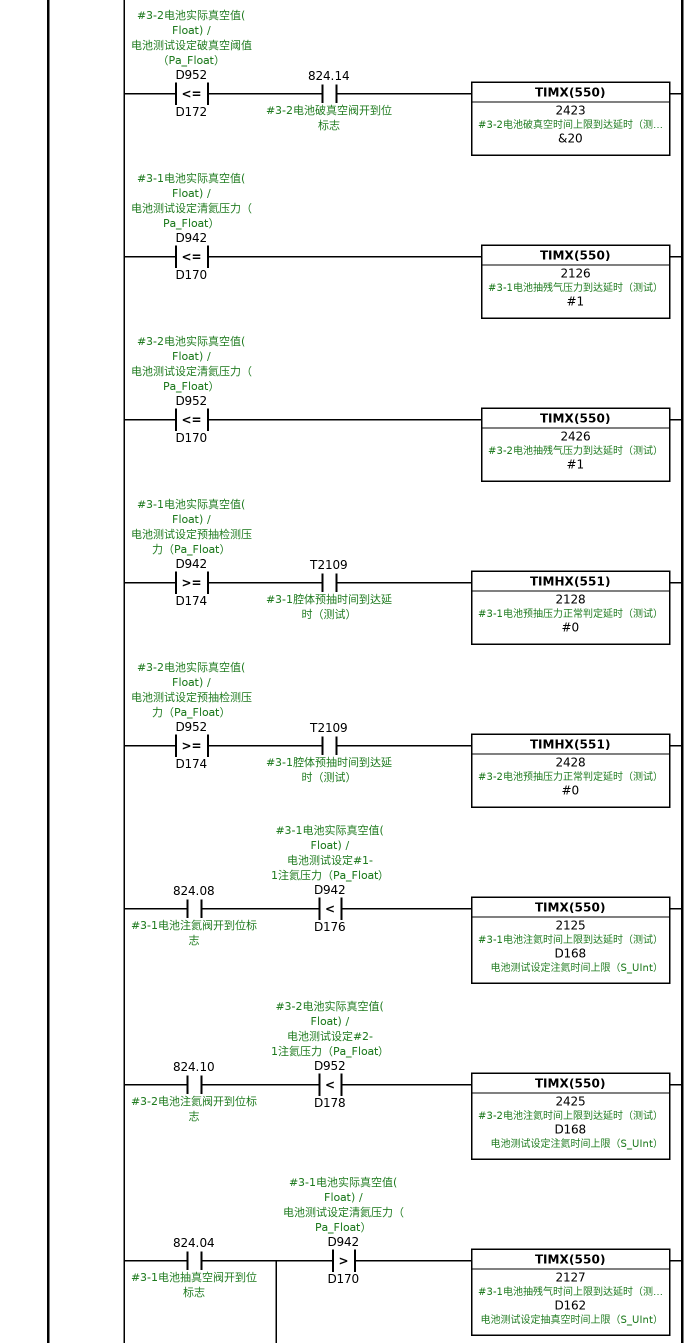

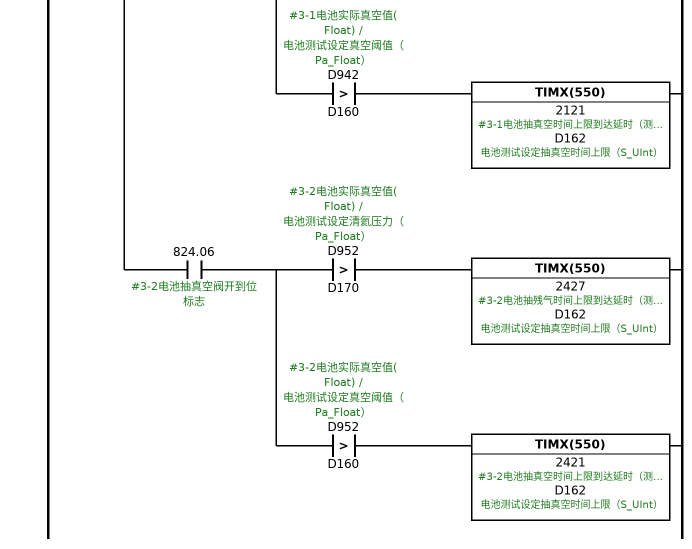
; rung 16
LD P_On
OUT TR0
AND<=F(332) D942 D160  ; #3-1电池实际真空值(Float), 电池测试设定真空阈值（Pa_Float）
LD 824.04  ; #3-1电池抽真空阀开到位标志
OR P_On
ANDLD
TIMX(550) 2120 #1  ; #3-1电池抽真空阈值到达延时（测试）
LD TR0
AND<=F(332) D952 D160  ; #3-2电池实际真空值(Float), 电池测试设定真空阈值（Pa_Float）
LD 824.06  ; #3-2电池抽真空阀开到位标志
OR P_On
ANDLD
TIMX(550) 2420 #1  ; #3-2电池抽真空阈值到达延时（测试）
LD TR0
LD>F(333) D942 D172  ; #3-1电池实际真空值(Float), 电池测试设定破真空阈值（Pa_Float）
OR H5.15  ; 腔体模式（0-正压 1-负压）
ANDLD
TIMX(550) 2122 #1  ; #3-1电池破真空阈值到达延时（测试）
LD TR0
LD>F(333) D952 D172  ; #3-2电池实际真空值(Float), 电池测试设定破真空阈值（Pa_Float）
OR H5.15  ; 腔体模式（0-正压 1-负压）
ANDLD
TIMX(550) 2422 #1  ; #3-2电池破真空阈值到达延时（测试）
LD TR0
AND>=F(334) D942 D176  ; #3-1电池实际真空值(Float), 电池测试设定#1-1注氦压力（Pa_Float）
AND 824.08  ; #3-1电池注氦阀开到位标志
TIMHX(551) 2124 #0  ; #3-1电池注氦压力到达延时（测试）
LD TR0
AND>=F(334) D952 D176  ; #3-2电池实际真空值(Float), 电池测试设定#1-1注氦压力（Pa_Float）
AND 824.10  ; #3-2电池注氦阀开到位标志
TIMHX(551) 2424 #0  ; #3-2电池注氦压力到达延时（测试）
LD TR0
AND<=F(332) D942 D172  ; #3-1电池实际真空值(Float), 电池测试设定破真空阈值（Pa_Float）
AND 824.12  ; #3-1电池破真空阀开到位标志
TIMX(550) 2123 &20  ; #3-1电池破真空时间上限到达延时（测试）
LD TR0
AND<=F(332) D952 D172  ; #3-2电池实际真空值(Float), 电池测试设定破真空阈值（Pa_Float）
AND 824.14  ; #3-2电池破真空阀开到位标志
TIMX(550) 2423 &20  ; #3-2电池破真空时间上限到达延时（测试）
LD TR0
AND<=F(332) D942 D170  ; #3-1电池实际真空值(Float), 电池测试设定清氦压力（Pa_Float）
TIMX(550) 2126 #1  ; #3-1电池抽残气压力到达延时（测试）
LD TR0
AND<=F(332) D952 D170  ; #3-2电池实际真空值(Float), 电池测试设定清氦压力（Pa_Float）
TIMX(550) 2426 #1  ; #3-2电池抽残气压力到达延时（测试）
LD TR0
AND>=F(334) D942 D174  ; #3-1电池实际真空值(Float), 电池测试设定预抽检测压力（Pa_Float）
AND T2109  ; #3-1腔体预抽时间到达延时（测试）
TIMHX(551) 2128 #0  ; #3-1电池预抽压力正常判定延时（测试）
LD TR0
AND>=F(334) D952 D174  ; #3-2电池实际真空值(Float), 电池测试设定预抽检测压力（Pa_Float）
AND T2109  ; #3-1腔体预抽时间到达延时（测试）
TIMHX(551) 2428 #0  ; #3-2电池预抽压力正常判定延时（测试）
LD TR0
AND 824.08  ; #3-1电池注氦阀开到位标志
AND<F(331) D942 D176  ; #3-1电池实际真空值(Float), 电池测试设定#1-1注氦压力（Pa_Float）
TIMX(550) 2125 D168  ; 电池测试设定注氦时间上限（S_UInt）, #3-1电池注氦时间上限到达延时（测试）
LD TR0
AND 824.10  ; #3-2电池注氦阀开到位标志
AND<F(331) D952 D178  ; #3-2电池实际真空值(Float), 电池测试设定#2-1注氦压力（Pa_Float）
TIMX(550) 2425 D168  ; 电池测试设定注氦时间上限（S_UInt）, #3-2电池注氦时间上限到达延时（测试）
LD TR0
AND 824.04  ; #3-1电池抽真空阀开到位标志
OUT TR1
AND>F(333) D942 D170  ; #3-1电池实际真空值(Float), 电池测试设定清氦压力（Pa_Float）
TIMX(550) 2127 D162  ; 电池测试设定抽真空时间上限（S_UInt）, #3-1电池抽残气时间上限到达延时（测试）
LD TR1
AND>F(333) D942 D160  ; #3-1电池实际真空值(Float), 电池测试设定真空阈值（Pa_Float）
TIMX(550) 2121 D162  ; 电池测试设定抽真空时间上限（S_UInt）, #3-1电池抽真空时间上限到达延时（测试）
LD TR0
AND 824.06  ; #3-2电池抽真空阀开到位标志
OUT TR0
AND>F(333) D952 D170  ; #3-2电池实际真空值(Float), 电池测试设定清氦压力（Pa_Float）
TIMX(550) 2427 D162  ; 电池测试设定抽真空时间上限（S_UInt）, #3-2电池抽残气时间上限到达延时（测试）
LD TR0
AND>F(333) D952 D160  ; #3-2电池实际真空值(Float), 电池测试设定真空阈值（Pa_Float）
TIMX(550) 2421 D162  ; 电池测试设定抽真空时间上限（S_UInt）, #3-2电池抽真空时间上限到达延时（测试）

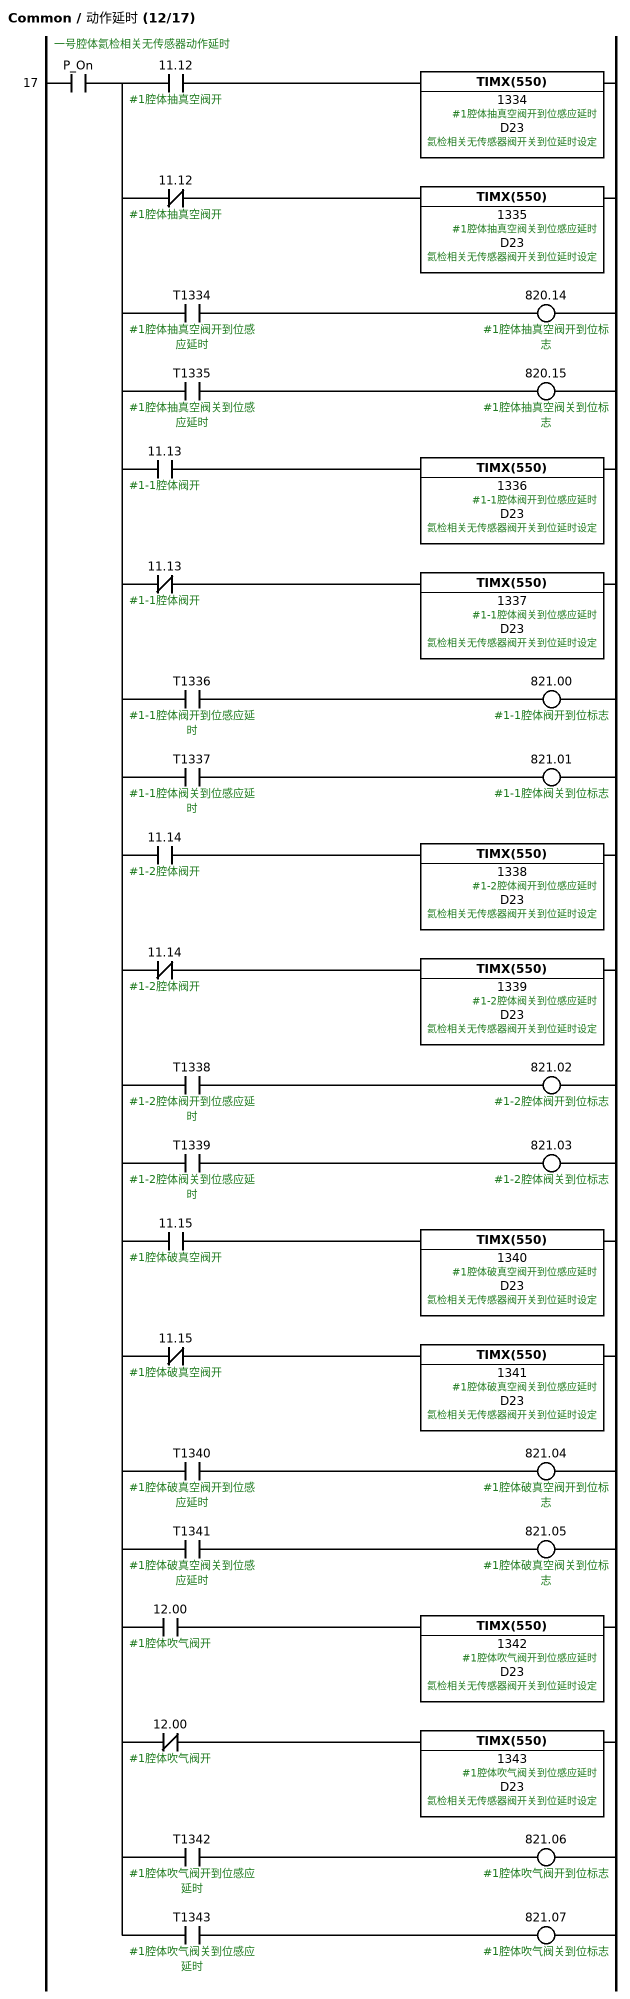
; rung 17: 一号腔体氦检相关无传感器动作延时
LD P_On
OUT TR0
AND 11.12  ; #1腔体抽真空阀开
TIMX(550) 1334 D23  ; 氦检相关无传感器阀开关到位延时设定, #1腔体抽真空阀开到位感应延时
LD TR0
ANDNOT 11.12  ; #1腔体抽真空阀开
TIMX(550) 1335 D23  ; 氦检相关无传感器阀开关到位延时设定, #1腔体抽真空阀关到位感应延时
LD TR0
AND T1334  ; #1腔体抽真空阀开到位感应延时
OUT 820.14  ; #1腔体抽真空阀开到位标志
LD TR0
AND T1335  ; #1腔体抽真空阀关到位感应延时
OUT 820.15  ; #1腔体抽真空阀关到位标志
LD TR0
AND 11.13  ; #1-1腔体阀开
TIMX(550) 1336 D23  ; 氦检相关无传感器阀开关到位延时设定, #1-1腔体阀开到位感应延时
LD TR0
ANDNOT 11.13  ; #1-1腔体阀开
TIMX(550) 1337 D23  ; 氦检相关无传感器阀开关到位延时设定, #1-1腔体阀关到位感应延时
LD TR0
AND T1336  ; #1-1腔体阀开到位感应延时
OUT 821.00  ; #1-1腔体阀开到位标志
LD TR0
AND T1337  ; #1-1腔体阀关到位感应延时
OUT 821.01  ; #1-1腔体阀关到位标志
LD TR0
AND 11.14  ; #1-2腔体阀开
TIMX(550) 1338 D23  ; 氦检相关无传感器阀开关到位延时设定, #1-2腔体阀开到位感应延时
LD TR0
ANDNOT 11.14  ; #1-2腔体阀开
TIMX(550) 1339 D23  ; 氦检相关无传感器阀开关到位延时设定, #1-2腔体阀关到位感应延时
LD TR0
AND T1338  ; #1-2腔体阀开到位感应延时
OUT 821.02  ; #1-2腔体阀开到位标志
LD TR0
AND T1339  ; #1-2腔体阀关到位感应延时
OUT 821.03  ; #1-2腔体阀关到位标志
LD TR0
AND 11.15  ; #1腔体破真空阀开
TIMX(550) 1340 D23  ; 氦检相关无传感器阀开关到位延时设定, #1腔体破真空阀开到位感应延时
LD TR0
ANDNOT 11.15  ; #1腔体破真空阀开
TIMX(550) 1341 D23  ; 氦检相关无传感器阀开关到位延时设定, #1腔体破真空阀关到位感应延时
LD TR0
AND T1340  ; #1腔体破真空阀开到位感应延时
OUT 821.04  ; #1腔体破真空阀开到位标志
LD TR0
AND T1341  ; #1腔体破真空阀关到位感应延时
OUT 821.05  ; #1腔体破真空阀关到位标志
LD TR0
AND 12.00  ; #1腔体吹气阀开
TIMX(550) 1342 D23  ; 氦检相关无传感器阀开关到位延时设定, #1腔体吹气阀开到位感应延时
LD TR0
ANDNOT 12.00  ; #1腔体吹气阀开
TIMX(550) 1343 D23  ; 氦检相关无传感器阀开关到位延时设定, #1腔体吹气阀关到位感应延时
LD TR0
AND T1342  ; #1腔体吹气阀开到位感应延时
OUT 821.06  ; #1腔体吹气阀开到位标志
LD TR0
AND T1343  ; #1腔体吹气阀关到位感应延时
OUT 821.07  ; #1腔体吹气阀关到位标志

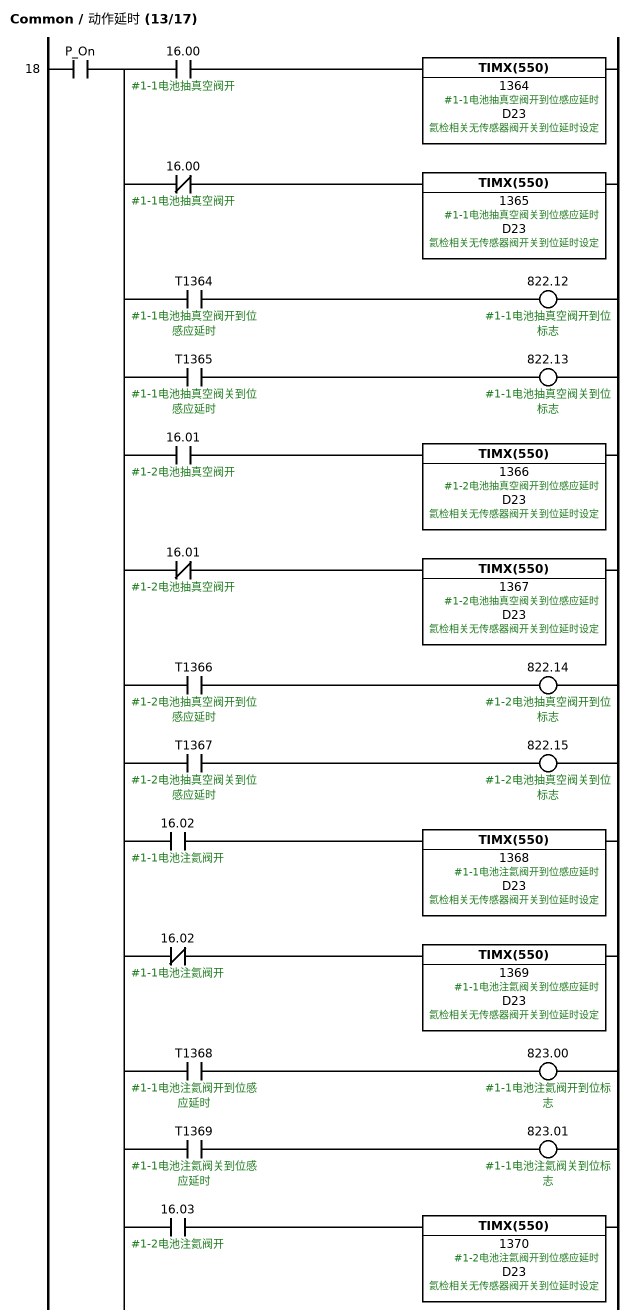

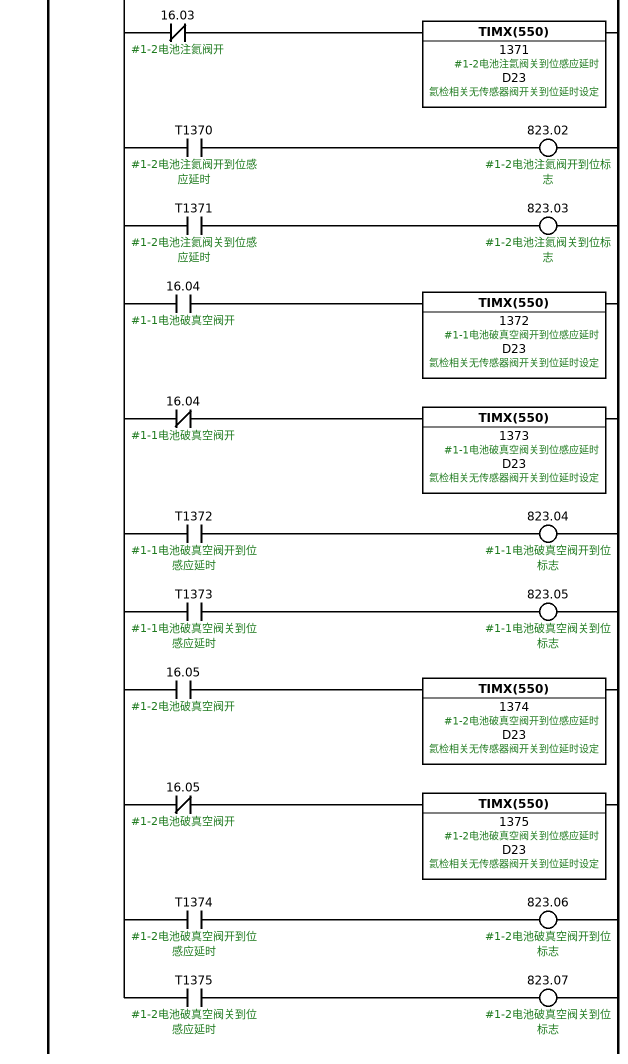
; rung 18
LD P_On
OUT TR0
AND 16.00  ; #1-1电池抽真空阀开
TIMX(550) 1364 D23  ; 氦检相关无传感器阀开关到位延时设定, #1-1电池抽真空阀开到位感应延时
LD TR0
ANDNOT 16.00  ; #1-1电池抽真空阀开
TIMX(550) 1365 D23  ; 氦检相关无传感器阀开关到位延时设定, #1-1电池抽真空阀关到位感应延时
LD TR0
AND T1364  ; #1-1电池抽真空阀开到位感应延时
OUT 822.12  ; #1-1电池抽真空阀开到位标志
LD TR0
AND T1365  ; #1-1电池抽真空阀关到位感应延时
OUT 822.13  ; #1-1电池抽真空阀关到位标志
LD TR0
AND 16.01  ; #1-2电池抽真空阀开
TIMX(550) 1366 D23  ; 氦检相关无传感器阀开关到位延时设定, #1-2电池抽真空阀开到位感应延时
LD TR0
ANDNOT 16.01  ; #1-2电池抽真空阀开
TIMX(550) 1367 D23  ; 氦检相关无传感器阀开关到位延时设定, #1-2电池抽真空阀关到位感应延时
LD TR0
AND T1366  ; #1-2电池抽真空阀开到位感应延时
OUT 822.14  ; #1-2电池抽真空阀开到位标志
LD TR0
AND T1367  ; #1-2电池抽真空阀关到位感应延时
OUT 822.15  ; #1-2电池抽真空阀关到位标志
LD TR0
AND 16.02  ; #1-1电池注氦阀开
TIMX(550) 1368 D23  ; 氦检相关无传感器阀开关到位延时设定, #1-1电池注氦阀开到位感应延时
LD TR0
ANDNOT 16.02  ; #1-1电池注氦阀开
TIMX(550) 1369 D23  ; 氦检相关无传感器阀开关到位延时设定, #1-1电池注氦阀关到位感应延时
LD TR0
AND T1368  ; #1-1电池注氦阀开到位感应延时
OUT 823.00  ; #1-1电池注氦阀开到位标志
LD TR0
AND T1369  ; #1-1电池注氦阀关到位感应延时
OUT 823.01  ; #1-1电池注氦阀关到位标志
LD TR0
AND 16.03  ; #1-2电池注氦阀开
TIMX(550) 1370 D23  ; 氦检相关无传感器阀开关到位延时设定, #1-2电池注氦阀开到位感应延时
LD TR0
ANDNOT 16.03  ; #1-2电池注氦阀开
TIMX(550) 1371 D23  ; 氦检相关无传感器阀开关到位延时设定, #1-2电池注氦阀关到位感应延时
LD TR0
AND T1370  ; #1-2电池注氦阀开到位感应延时
OUT 823.02  ; #1-2电池注氦阀开到位标志
LD TR0
AND T1371  ; #1-2电池注氦阀关到位感应延时
OUT 823.03  ; #1-2电池注氦阀关到位标志
LD TR0
AND 16.04  ; #1-1电池破真空阀开
TIMX(550) 1372 D23  ; 氦检相关无传感器阀开关到位延时设定, #1-1电池破真空阀开到位感应延时
LD TR0
ANDNOT 16.04  ; #1-1电池破真空阀开
TIMX(550) 1373 D23  ; 氦检相关无传感器阀开关到位延时设定, #1-1电池破真空阀关到位感应延时
LD TR0
AND T1372  ; #1-1电池破真空阀开到位感应延时
OUT 823.04  ; #1-1电池破真空阀开到位标志
LD TR0
AND T1373  ; #1-1电池破真空阀关到位感应延时
OUT 823.05  ; #1-1电池破真空阀关到位标志
LD TR0
AND 16.05  ; #1-2电池破真空阀开
TIMX(550) 1374 D23  ; 氦检相关无传感器阀开关到位延时设定, #1-2电池破真空阀开到位感应延时
LD TR0
ANDNOT 16.05  ; #1-2电池破真空阀开
TIMX(550) 1375 D23  ; 氦检相关无传感器阀开关到位延时设定, #1-2电池破真空阀关到位感应延时
LD TR0
AND T1374  ; #1-2电池破真空阀开到位感应延时
OUT 823.06  ; #1-2电池破真空阀开到位标志
LD TR0
AND T1375  ; #1-2电池破真空阀关到位感应延时
OUT 823.07  ; #1-2电池破真空阀关到位标志

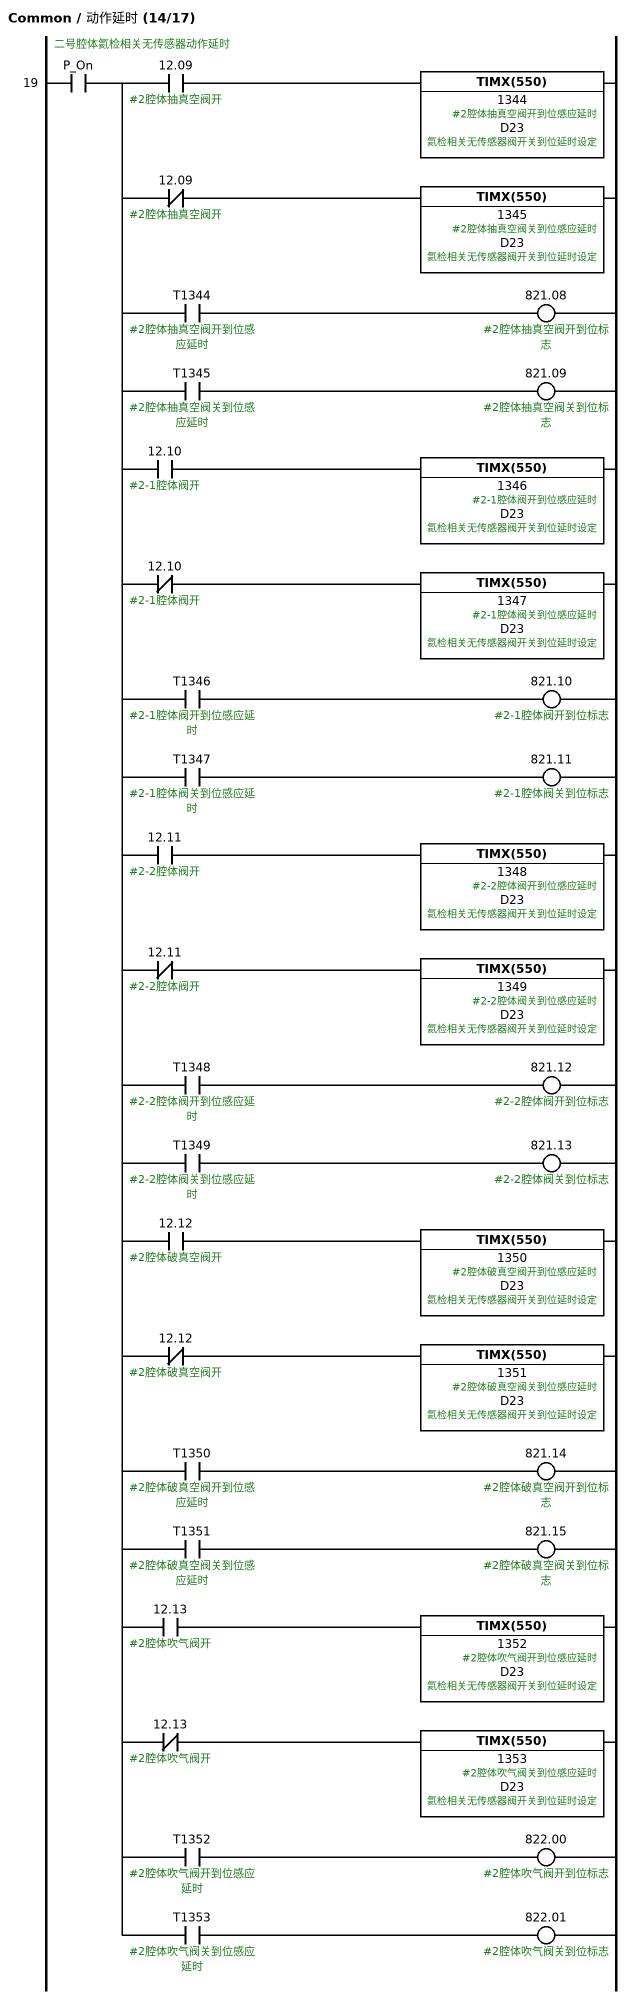
; rung 19: 二号腔体氦检相关无传感器动作延时
LD P_On
OUT TR0
AND 12.09  ; #2腔体抽真空阀开
TIMX(550) 1344 D23  ; 氦检相关无传感器阀开关到位延时设定, #2腔体抽真空阀开到位感应延时
LD TR0
ANDNOT 12.09  ; #2腔体抽真空阀开
TIMX(550) 1345 D23  ; 氦检相关无传感器阀开关到位延时设定, #2腔体抽真空阀关到位感应延时
LD TR0
AND T1344  ; #2腔体抽真空阀开到位感应延时
OUT 821.08  ; #2腔体抽真空阀开到位标志
LD TR0
AND T1345  ; #2腔体抽真空阀关到位感应延时
OUT 821.09  ; #2腔体抽真空阀关到位标志
LD TR0
AND 12.10  ; #2-1腔体阀开
TIMX(550) 1346 D23  ; 氦检相关无传感器阀开关到位延时设定, #2-1腔体阀开到位感应延时
LD TR0
ANDNOT 12.10  ; #2-1腔体阀开
TIMX(550) 1347 D23  ; 氦检相关无传感器阀开关到位延时设定, #2-1腔体阀关到位感应延时
LD TR0
AND T1346  ; #2-1腔体阀开到位感应延时
OUT 821.10  ; #2-1腔体阀开到位标志
LD TR0
AND T1347  ; #2-1腔体阀关到位感应延时
OUT 821.11  ; #2-1腔体阀关到位标志
LD TR0
AND 12.11  ; #2-2腔体阀开
TIMX(550) 1348 D23  ; 氦检相关无传感器阀开关到位延时设定, #2-2腔体阀开到位感应延时
LD TR0
ANDNOT 12.11  ; #2-2腔体阀开
TIMX(550) 1349 D23  ; 氦检相关无传感器阀开关到位延时设定, #2-2腔体阀关到位感应延时
LD TR0
AND T1348  ; #2-2腔体阀开到位感应延时
OUT 821.12  ; #2-2腔体阀开到位标志
LD TR0
AND T1349  ; #2-2腔体阀关到位感应延时
OUT 821.13  ; #2-2腔体阀关到位标志
LD TR0
AND 12.12  ; #2腔体破真空阀开
TIMX(550) 1350 D23  ; 氦检相关无传感器阀开关到位延时设定, #2腔体破真空阀开到位感应延时
LD TR0
ANDNOT 12.12  ; #2腔体破真空阀开
TIMX(550) 1351 D23  ; 氦检相关无传感器阀开关到位延时设定, #2腔体破真空阀关到位感应延时
LD TR0
AND T1350  ; #2腔体破真空阀开到位感应延时
OUT 821.14  ; #2腔体破真空阀开到位标志
LD TR0
AND T1351  ; #2腔体破真空阀关到位感应延时
OUT 821.15  ; #2腔体破真空阀关到位标志
LD TR0
AND 12.13  ; #2腔体吹气阀开
TIMX(550) 1352 D23  ; 氦检相关无传感器阀开关到位延时设定, #2腔体吹气阀开到位感应延时
LD TR0
ANDNOT 12.13  ; #2腔体吹气阀开
TIMX(550) 1353 D23  ; 氦检相关无传感器阀开关到位延时设定, #2腔体吹气阀关到位感应延时
LD TR0
AND T1352  ; #2腔体吹气阀开到位感应延时
OUT 822.00  ; #2腔体吹气阀开到位标志
LD TR0
AND T1353  ; #2腔体吹气阀关到位感应延时
OUT 822.01  ; #2腔体吹气阀关到位标志

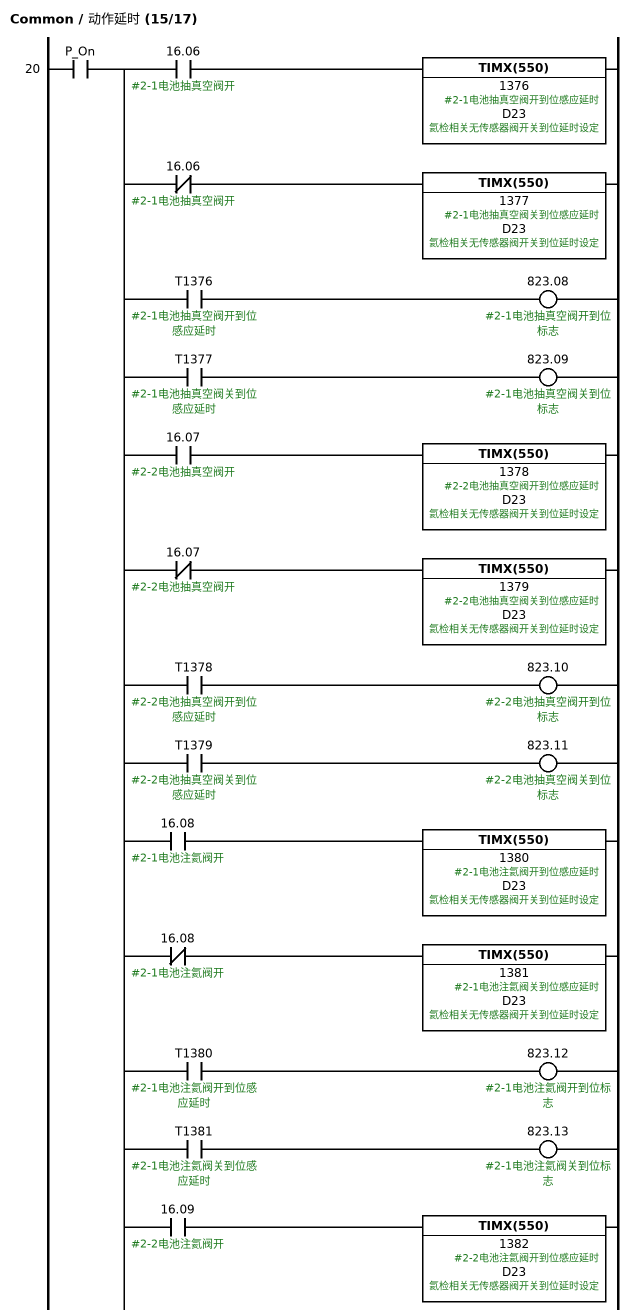

